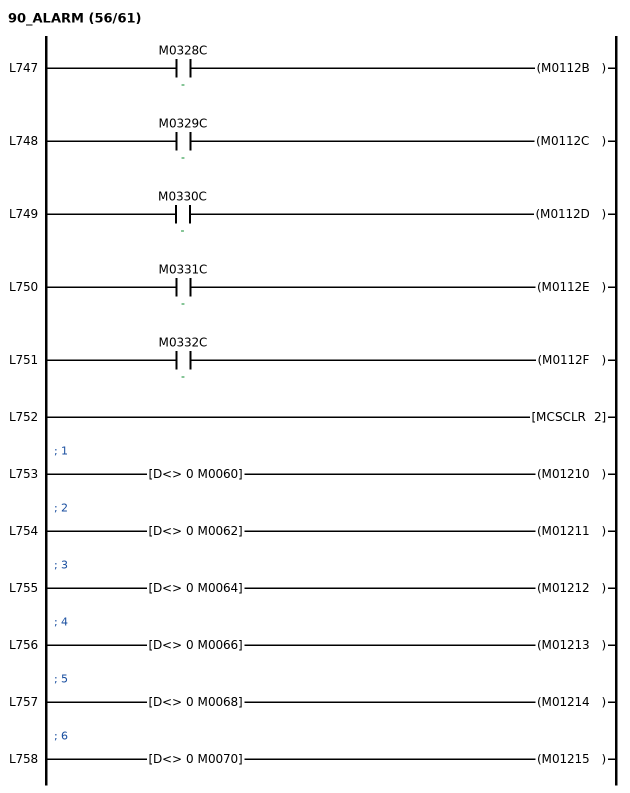
[picture p432: 90_ALARM rungs L747-L758]
; L747
LOAD      M0328C	// -
OUT       M0112B
; L748
LOAD      M0329C	// -
OUT       M0112C
; L749
LOAD      M0330C	// -
OUT       M0112D
; L750
LOAD      M0331C	// -
OUT       M0112E
; L751
LOAD      M0332C	// -
OUT       M0112F
; L752
MCSCLR    2
; L753
LOADD<>   0 M0060
OUT       M01210
// output comment: 1
; L754
LOADD<>   0 M0062
OUT       M01211
// output comment: 2
; L755
LOADD<>   0 M0064
OUT       M01212
// output comment: 3
; L756
LOADD<>   0 M0066
OUT       M01213
// output comment: 4
; L757
LOADD<>   0 M0068
OUT       M01214
// output comment: 5
; L758
LOADD<>   0 M0070
OUT       M01215
// output comment: 6

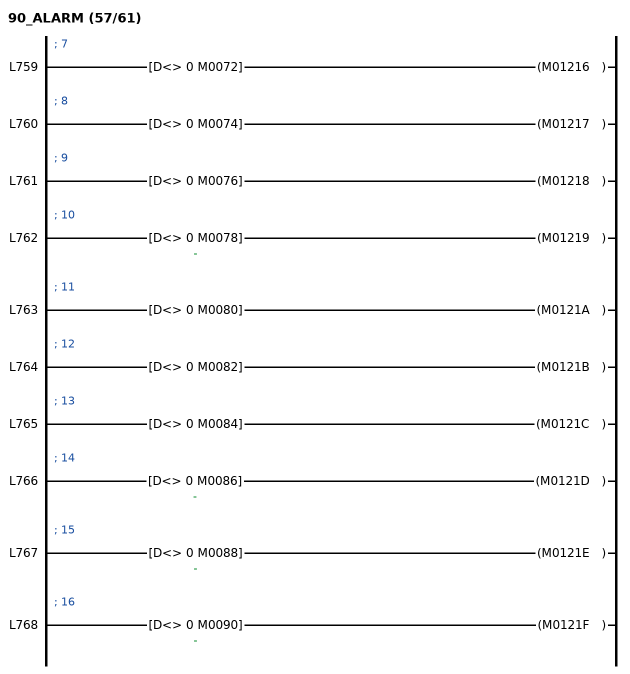
; L759
LOADD<>   0 M0072
OUT       M01216
// output comment: 7
; L760
LOADD<>   0 M0074
OUT       M01217
// output comment: 8
; L761
LOADD<>   0 M0076
OUT       M01218
// output comment: 9
; L762
LOADD<>   0 M0078	// -
OUT       M01219
// output comment: 10
; L763
LOADD<>   0 M0080
OUT       M0121A
// output comment: 11
; L764
LOADD<>   0 M0082
OUT       M0121B
// output comment: 12
; L765
LOADD<>   0 M0084
OUT       M0121C
// output comment: 13
; L766
LOADD<>   0 M0086	// -
OUT       M0121D
// output comment: 14
; L767
LOADD<>   0 M0088	// -
OUT       M0121E
// output comment: 15
; L768
LOADD<>   0 M0090	// -
OUT       M0121F
// output comment: 16

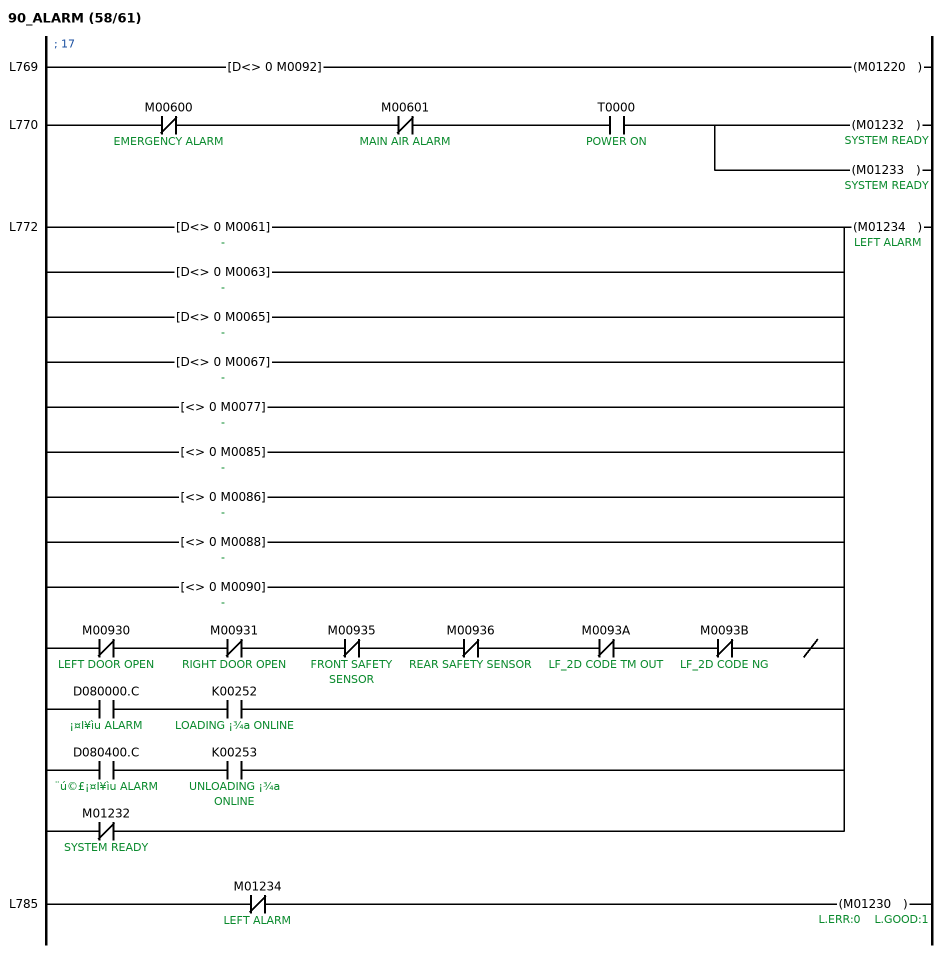
; L769
LOADD<>   0 M0092
OUT       M01220
// output comment: 17
; L770
LOAD NOT  M00600	// EMERGENCY ALARM
AND NOT   M00601	// MAIN AIR ALARM
AND       T0000	// POWER ON
OUT       M01232	// SYSTEM READY
OUT       M01233	// SYSTEM READY
; L772
LOADD<>   0 M0061	// -
ORD<>     0 M0063	// -
ORD<>     0 M0065	// -
ORD<>     0 M0067	// -
OR<>      0 M0077	// -
OR<>      0 M0085	// -
OR<>      0 M0086	// -
OR<>      0 M0088	// -
OR<>      0 M0090	// -
LOAD NOT  M00930	// LEFT DOOR OPEN
AND NOT   M00931	// RIGHT DOOR OPEN
AND NOT   M00935	// FRONT SAFETY SENSOR
AND NOT   M00936	// REAR SAFETY SENSOR
AND NOT   M0093A	// LF_2D CODE TM OUT
AND NOT   M0093B	// LF_2D CODE NG
NOT
OR LOAD
LOAD      D080000.C	// ¡¤I¥ìu ALARM
AND       K00252	// LOADING ¡¾a ONLINE
OR LOAD
LOAD      D080400.C	// ¨ú©£¡¤I¥ìu ALARM
AND       K00253	// UNLOADING ¡¾a ONLINE
OR LOAD
OR NOT    M01232	// SYSTEM READY
OUT       M01234	// LEFT ALARM
; L785
LOAD NOT  M01234	// LEFT ALARM
OUT       M01230	// L.ERR:0    L.GOOD:1

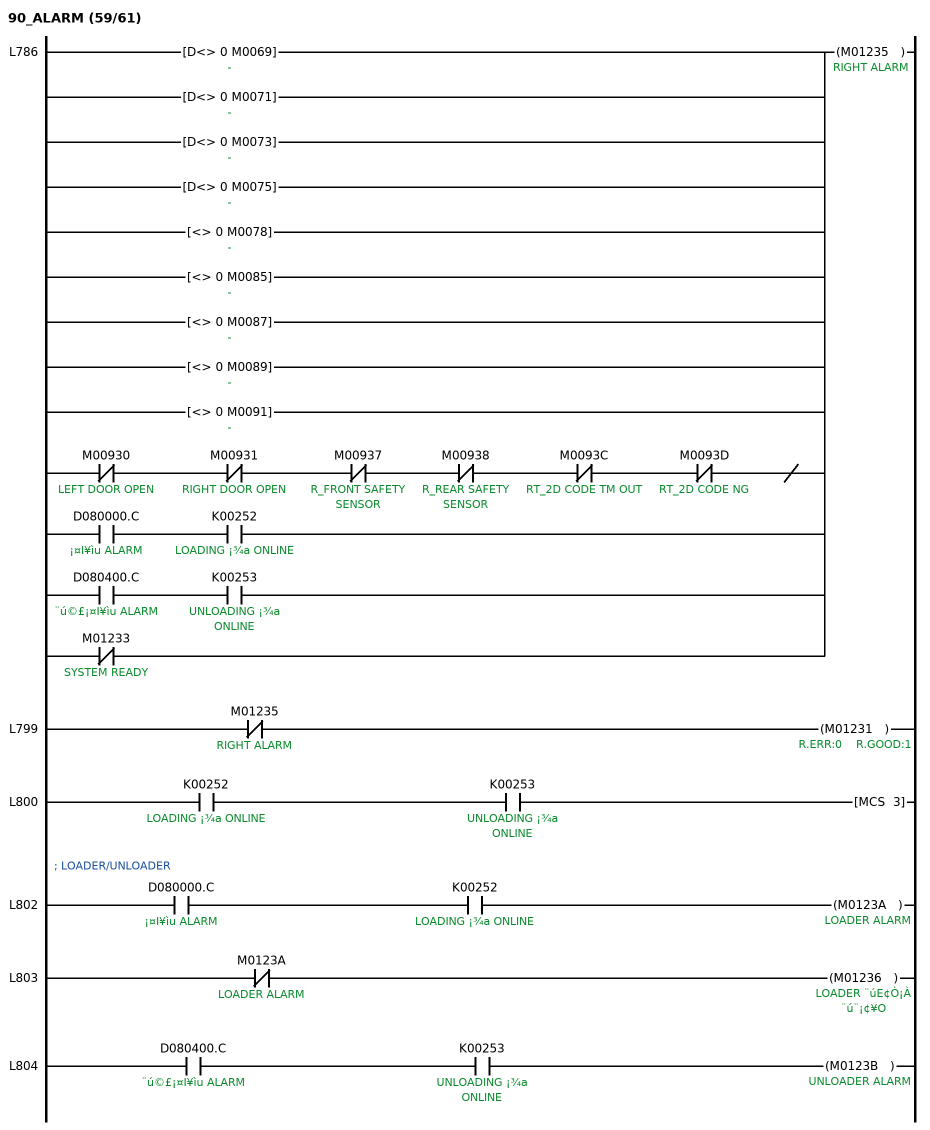
; L786
LOADD<>   0 M0069	// -
ORD<>     0 M0071	// -
ORD<>     0 M0073	// -
ORD<>     0 M0075	// -
OR<>      0 M0078	// -
OR<>      0 M0085	// -
OR<>      0 M0087	// -
OR<>      0 M0089	// -
OR<>      0 M0091	// -
LOAD NOT  M00930	// LEFT DOOR OPEN
AND NOT   M00931	// RIGHT DOOR OPEN
AND NOT   M00937	// R_FRONT SAFETY SENSOR
AND NOT   M00938	// R_REAR SAFETY SENSOR
AND NOT   M0093C	// RT_2D CODE TM OUT
AND NOT   M0093D	// RT_2D CODE NG
NOT
OR LOAD
LOAD      D080000.C	// ¡¤I¥ìu ALARM
AND       K00252	// LOADING ¡¾a ONLINE
OR LOAD
LOAD      D080400.C	// ¨ú©£¡¤I¥ìu ALARM
AND       K00253	// UNLOADING ¡¾a ONLINE
OR LOAD
OR NOT    M01233	// SYSTEM READY
OUT       M01235	// RIGHT ALARM
; L799
LOAD NOT  M01235	// RIGHT ALARM
OUT       M01231	// R.ERR:0    R.GOOD:1
; L800
LOAD      K00252	// LOADING ¡¾a ONLINE
AND       K00253	// UNLOADING ¡¾a ONLINE
MCS       3
// LOADER/UNLOADER
; L802
LOAD      D080000.C	// ¡¤I¥ìu ALARM
AND       K00252	// LOADING ¡¾a ONLINE
OUT       M0123A	// LOADER ALARM
; L803
LOAD NOT  M0123A	// LOADER ALARM
OUT       M01236	// LOADER ¨úE¢Ò¡À ¨ú¨¡¢¥O
; L804
LOAD      D080400.C	// ¨ú©£¡¤I¥ìu ALARM
AND       K00253	// UNLOADING ¡¾a ONLINE
OUT       M0123B	// UNLOADER ALARM

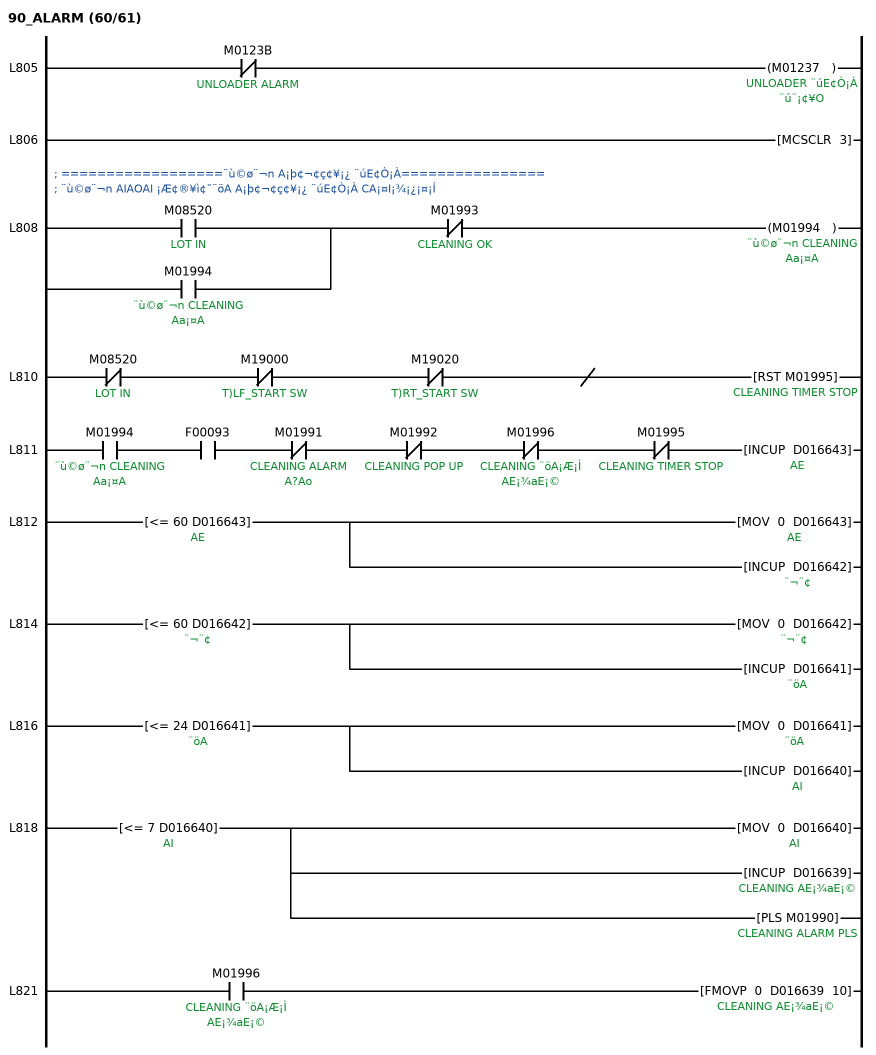
; L805
LOAD NOT  M0123B	// UNLOADER ALARM
OUT       M01237	// UNLOADER ¨úE¢Ò¡À ¨ú¨¡¢¥O
; L806
MCSCLR    3
// ==================¨ù©ø¨¬n A¡þ¢¬¢ç¢¥¡¿ ¨úE¢Ò¡À================
; L808
LOAD      M08520	// LOT IN
OR        M01994	// ¨ù©ø¨¬n CLEANING Aa¡¤A
AND NOT   M01993	// CLEANING OK
OUT       M01994	// ¨ù©ø¨¬n CLEANING Aa¡¤A
// output comment: ¨ù©ø¨¬n AIAOAI ¡Æ¢®¥ì¢¯¨öA A¡þ¢¬¢ç¢¥¡¿ ¨úE¢Ò¡À CA¡¤I¡¾¡¿¡¤¡Í
; L810
LOAD NOT  M08520	// LOT IN
AND NOT   M19000	// T)LF_START SW
AND NOT   M19020	// T)RT_START SW
NOT
RST       M01995	// CLEANING TIMER STOP
; L811
LOAD      M01994	// ¨ù©ø¨¬n CLEANING Aa¡¤A
AND       F00093
AND NOT   M01991	// CLEANING ALARM A?Ao
AND NOT   M01992	// CLEANING POP UP
AND NOT   M01996	// CLEANING ¨öA¡Æ¡Ì AE¡¾aE¡©
AND NOT   M01995	// CLEANING TIMER STOP
INCUP     D016643	// AE
; L812
LOAD<=    60 D016643	// AE
MOV       0 D016643	// AE
INCUP     D016642	// ¨¬¨¢
; L814
LOAD<=    60 D016642	// ¨¬¨¢
MOV       0 D016642	// ¨¬¨¢
INCUP     D016641	// ¨öA
; L816
LOAD<=    24 D016641	// ¨öA
MOV       0 D016641	// ¨öA
INCUP     D016640	// AI
; L818
LOAD<=    7 D016640	// AI
MOV       0 D016640	// AI
INCUP     D016639	// CLEANING AE¡¾aE¡©
OUTP      M01990	// CLEANING ALARM PLS
; L821
LOAD      M01996	// CLEANING ¨öA¡Æ¡Ì AE¡¾aE¡©
FMOVP     0 D016639 10	// CLEANING AE¡¾aE¡©

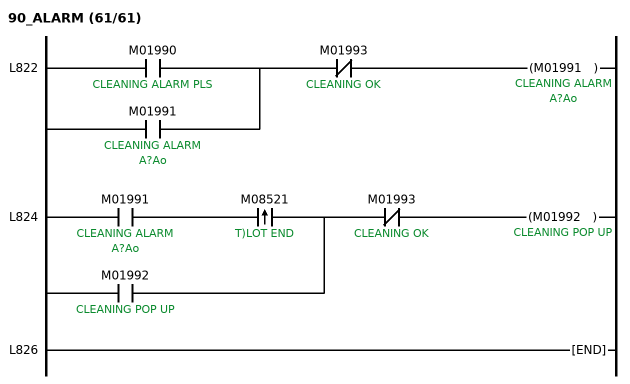
; L822
LOAD      M01990	// CLEANING ALARM PLS
OR        M01991	// CLEANING ALARM A?Ao
AND NOT   M01993	// CLEANING OK
OUT       M01991	// CLEANING ALARM A?Ao
; L824
LOAD      M01991	// CLEANING ALARM A?Ao
ANDP      M08521	// T)LOT END
OR        M01992	// CLEANING POP UP
AND NOT   M01993	// CLEANING OK
OUT       M01992	// CLEANING POP UP
; L826
END

PROGRAM 91_DEVICE_CHANGE (task: ¨ö¨¬A¥ì CA¡¤I¡¾¡¿¡¤¡Í)

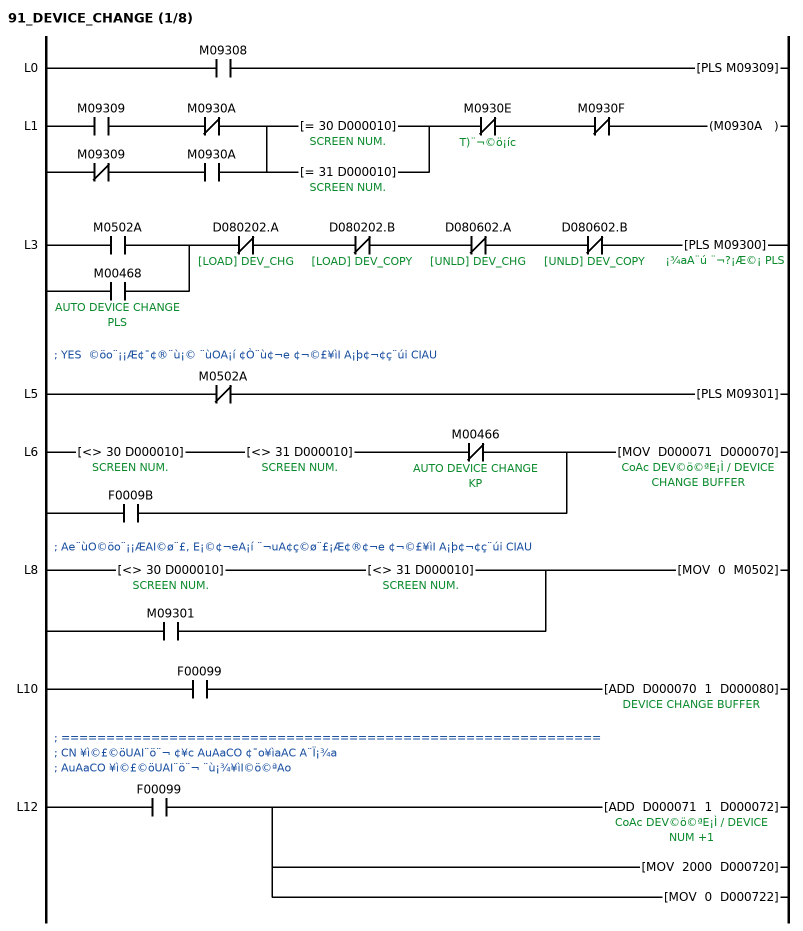
; L0
LOAD      M09308
OUTP      M09309
; L1
LOAD      M09309
AND NOT   M0930A
LOAD NOT  M09309
AND       M0930A
OR LOAD
LOAD=     30 D000010	// SCREEN NUM.
OR=       31 D000010	// SCREEN NUM.
AND LOAD
AND NOT   M0930E	// T)¨¬©ö¡íc
AND NOT   M0930F
OUT       M0930A
; L3
LOAD      M0502A
OR        M00468	// AUTO DEVICE CHANGE PLS
AND NOT   D080202.A	// [LOAD] DEV_CHG
AND NOT   D080202.B	// [LOAD] DEV_COPY
AND NOT   D080602.A	// [UNLD] DEV_CHG
AND NOT   D080602.B	// [UNLD] DEV_COPY
OUTP      M09300	// ¡¾aA¨ú ¨¬?¡Æ©¡ PLS
; L5
LOAD NOT  M0502A
OUTP      M09301
// output comment: YES  ©öo¨¡¡Æ¢¯¢®¨ù¡© ¨ùOA¡í ¢Ò¨ù¢¬e ¢¬©£¥ìI A¡þ¢¬¢ç¨úi CIAU
; L6
LOAD<>    30 D000010	// SCREEN NUM.
AND<>     31 D000010	// SCREEN NUM.
AND NOT   M00466	// AUTO DEVICE CHANGE KP
OR        F0009B
MOV       D000071 D000070	// CoAc DEV©ö©ªE¡Ì / DEVICE CHANGE BUFFER
; L8
LOAD<>    30 D000010	// SCREEN NUM.
AND<>     31 D000010	// SCREEN NUM.
OR        M09301
MOV       0 M0502
// output comment: Ae¨ùO©öo¨¡¡ÆAI©ø¨£, E¡©¢¬eA¡í ¨¬uA¢ç©ø¨£¡Æ¢®¢¬e ¢¬©£¥ìI A¡þ¢¬¢ç¨úi CIAU
; L10
LOAD      F00099
ADD       D000070 1 D000080	// DEVICE CHANGE BUFFER
// ============================================================
; L12
LOAD      F00099
ADD       D000071 1 D000072	// CoAc DEV©ö©ªE¡Ì / DEVICE NUM +1
MOV       2000 D000720
MOV       0 D000722
// output comment: CN ¥ì©£©öUAI¨ö¨¬ ¢¥c AuAaCO ¢¯o¥ìaAC A¨Ï¡¾a
// output comment: AuAaCO ¥ì©£©öUAI¨ö¨¬ ¨ù¡¾¥ìI©ö©ªAo

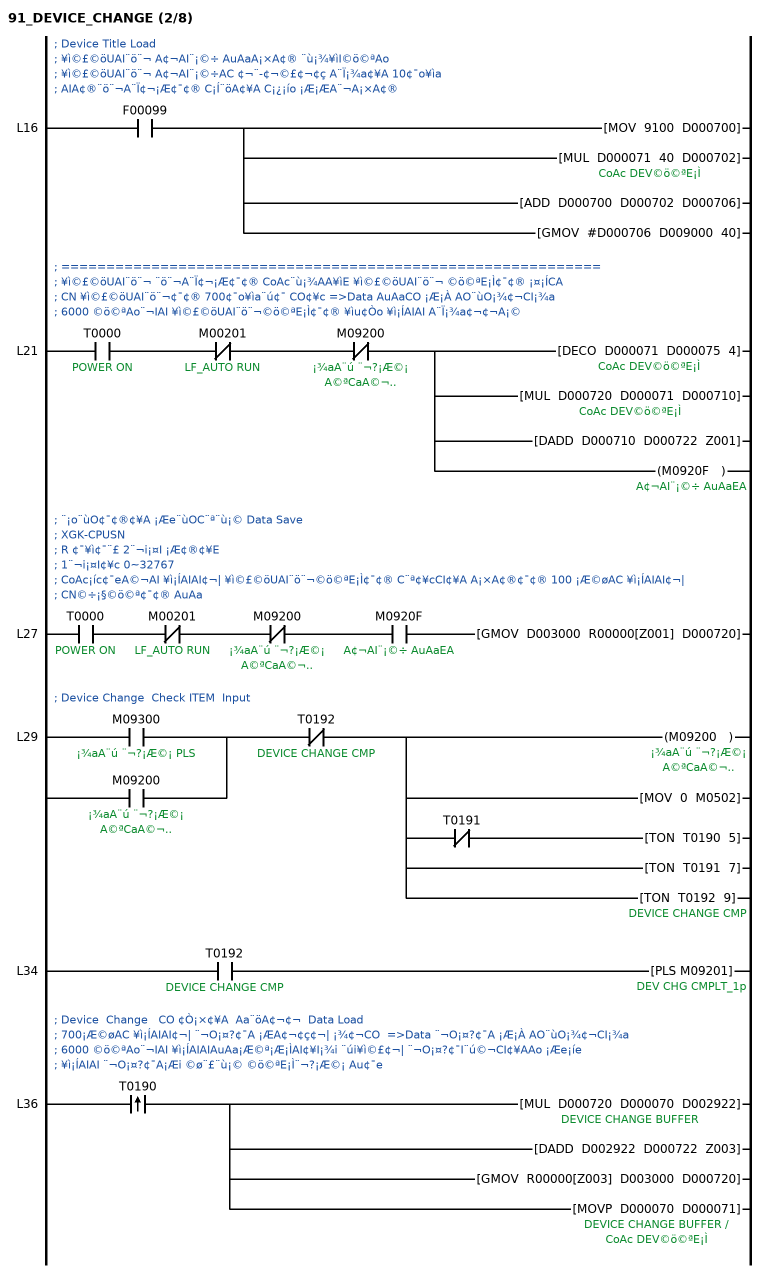
// Device Title Load
; L16
LOAD      F00099
MOV       9100 D000700
MUL       D000071 40 D000702	// CoAc DEV©ö©ªE¡Ì
ADD       D000700 D000702 D000706
GMOV      #D000706 D009000 40
// output comment: ¥ì©£©öUAI¨ö¨¬ A¢¬AI¨¡©÷ AuAaA¡×A¢® ¨ù¡¾¥ìI©ö©ªAo
// output comment: ¥ì©£©öUAI¨ö¨¬ A¢¬AI¨¡©÷AC ¢¬¨­¢¬©£¢¬¢ç A¨Ï¡¾a¢¥A 10¢¯o¥ìa
// output comment: AIA¢®¨ö¨¬A¨Ï¢¬¡Æ¢¯¢® C¡Í¨öA¢¥A C¡¿¡ío ¡Æ¡ÆA¨¬A¡×A¢®
// ============================================================
; L21
LOAD      T0000	// POWER ON
AND NOT   M00201	// LF_AUTO RUN
AND NOT   M09200	// ¡¾aA¨ú ¨¬?¡Æ©¡ A©ªCaA©¬..
DECO      D000071 D000075 4	// CoAc DEV©ö©ªE¡Ì
MUL       D000720 D000071 D000710	// CoAc DEV©ö©ªE¡Ì
DADD      D000710 D000722 Z001
OUT       M0920F	// A¢¬AI¨¡©÷ AuAaEA
// output comment: ¥ì©£©öUAI¨ö¨¬ ¨ö¨¬A¨Ï¢¬¡Æ¢¯¢® CoAc¨ù¡¾AA¥ìE ¥ì©£©öUAI¨ö¨¬ ©ö©ªE¡Ì¢¯¢® ¡¤¡ÍCA
// output comment: CN ¥ì©£©öUAI¨ö¨¬¢¯¢® 700¢¯o¥ìa¨ú¢¯ CO¢¥c =>Data AuAaCO ¡Æ¡À AO¨ùO¡¾¢¬CI¡¾a
// output comment: 6000 ©ö©ªAo¨¬IAI ¥ì©£©öUAI¨ö¨¬©ö©ªE¡Ì¢¯¢® ¥ìu¢Òo ¥ì¡ÍAIAI A¨Ï¡¾a¢¬¢¬A¡©
// ¨¡o¨ùO¢¯¢®¢¥A ¡Æe¨ùOC¨ª¨ù¡© Data Save
// XGK-CPUSN
// R ¢¯¥ì¢¯¨£ 2¨¬i¡¤I ¡Æ¢®¢¥E
// 1¨¬i¡¤I¢¥c 0~32767
; L27
LOAD      T0000	// POWER ON
AND NOT   M00201	// LF_AUTO RUN
AND NOT   M09200	// ¡¾aA¨ú ¨¬?¡Æ©¡ A©ªCaA©¬..
AND       M0920F	// A¢¬AI¨¡©÷ AuAaEA
GMOV      D003000 R00000[Z001] D000720
// output comment: CoAc¡íc¢¯eA©¬AI ¥ì¡ÍAIAI¢¬| ¥ì©£©öUAI¨ö¨¬©ö©ªE¡Ì¢¯¢® C¨ª¢¥cCI¢¥A A¡×A¢®¢¯¢® 100 ¡Æ©øAC ¥ì¡ÍAIAI¢¬| CN©÷¡§©ö©ª¢¯¢® AuAa
// Device Change  Check ITEM  Input
; L29
LOAD      M09300	// ¡¾aA¨ú ¨¬?¡Æ©¡ PLS
OR        M09200	// ¡¾aA¨ú ¨¬?¡Æ©¡ A©ªCaA©¬..
AND NOT   T0192	// DEVICE CHANGE CMP
OUT       M09200	// ¡¾aA¨ú ¨¬?¡Æ©¡ A©ªCaA©¬..
MOV       0 M0502
MPUSH
AND NOT   T0191
TON       T0190 5
MPOP
TON       T0191 7
TON       T0192 9	// DEVICE CHANGE CMP
; L34
LOAD      T0192	// DEVICE CHANGE CMP
OUTP      M09201	// DEV CHG CMPLT_1p
// Device  Change   CO ¢Ò¡×¢¥A  Aa¨öA¢¬¢¬  Data Load
; L36
LOADP     T0190
MUL       D000720 D000070 D002922	// DEVICE CHANGE BUFFER
DADD      D002922 D000722 Z003
GMOV      R00000[Z003] D003000 D000720
MOVP      D000070 D000071	// DEVICE CHANGE BUFFER / CoAc DEV©ö©ªE¡Ì
// output comment: 700¡Æ©øAC ¥ì¡ÍAIAI¢¬| ¨¬O¡¤?¢¯A ¡ÆA¢¬¢ç¢¬| ¡¾¢¬CO  =>Data ¨¬O¡¤?¢¯A ¡Æ¡À AO¨ùO¡¾¢¬CI¡¾a
// output comment: 6000 ©ö©ªAo¨¬IAI ¥ì¡ÍAIAIAuAa¡Æ©ª¡Æ¡ÌAI¢¥I¡¾i ¨úi¥ì©£¢¬| ¨¬O¡¤?¢¯I¨ú©¬CI¢¥AAo ¡Æe¡íe
// output comment: ¥ì¡ÍAIAI ¨¬O¡¤?¢¯A¡Æi ©ø¨£¨ù¡© ©ö©ªE¡Ì¨¬?¡Æ©¡ Au¢¯e

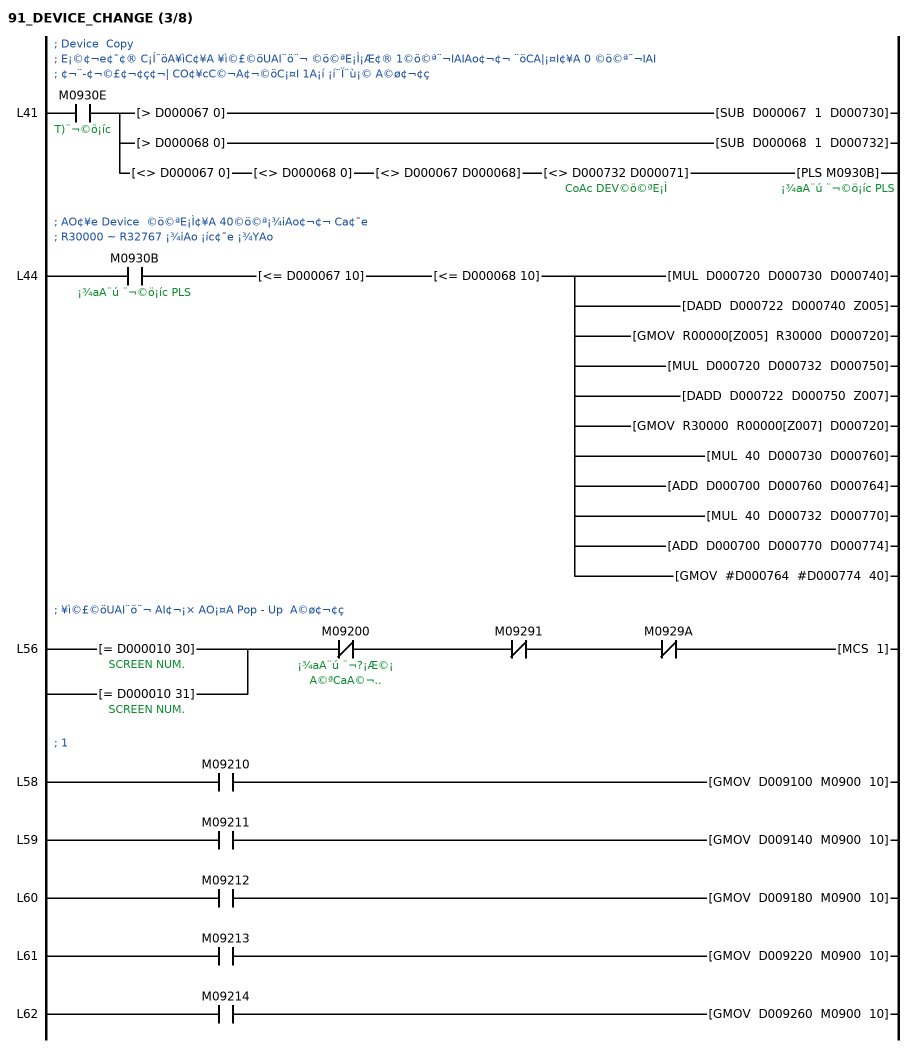
// Device  Copy
; L41
LOAD      M0930E	// T)¨¬©ö¡íc
MPUSH
AND>      D000067 0
SUB       D000067 1 D000730
MLOAD
AND>      D000068 0
SUB       D000068 1 D000732
MPOP
AND<>     D000067 0
AND<>     D000068 0
AND<>     D000067 D000068
AND<>     D000732 D000071	// CoAc DEV©ö©ªE¡Ì
OUTP      M0930B	// ¡¾aA¨ú ¨¬©ö¡íc PLS
// output comment: E¡©¢¬e¢¯¢® C¡Í¨öA¥ìC¢¥A ¥ì©£©öUAI¨ö¨¬ ©ö©ªE¡Ì¡Æ¢® 1©ö©ª¨¬IAIAo¢¬¢¬ ¨öCA|¡¤I¢¥A 0 ©ö©ª¨¬IAI
// output comment: ¢¬¨­¢¬©£¢¬¢ç¢¬| CO¢¥cC©¬A¢¬©öC¡¤I 1A¡í ¡í¨Ï¨ù¡© A©ø¢¬¢ç
; L44
LOAD      M0930B	// ¡¾aA¨ú ¨¬©ö¡íc PLS
AND<=     D000067 10
AND<=     D000068 10
MUL       D000720 D000730 D000740
DADD      D000722 D000740 Z005
GMOV      R00000[Z005] R30000 D000720
MUL       D000720 D000732 D000750
DADD      D000722 D000750 Z007
GMOV      R30000 R00000[Z007] D000720
MUL       40 D000730 D000760
ADD       D000700 D000760 D000764
MUL       40 D000732 D000770
ADD       D000700 D000770 D000774
GMOV      #D000764 #D000774 40
// output comment: AO¢¥e Device  ©ö©ªE¡Ì¢¥A 40©ö©ª¡¾iAo¢¬¢¬ Ca¢¯e
// output comment: R30000 ~ R32767 ¡¾iAo ¡íc¢¯e ¡¾YAo
// ¥ì©£©öUAI¨ö¨¬ AI¢¬¡× AO¡¤A Pop - Up  A©ø¢¬¢ç
; L56
LOAD=     D000010 30	// SCREEN NUM.
OR=       D000010 31	// SCREEN NUM.
AND NOT   M09200	// ¡¾aA¨ú ¨¬?¡Æ©¡ A©ªCaA©¬..
AND NOT   M09291
AND NOT   M0929A
MCS       1
; L58
LOAD      M09210
GMOV      D009100 M0900 10
// output comment: 1
; L59
LOAD      M09211
GMOV      D009140 M0900 10
; L60
LOAD      M09212
GMOV      D009180 M0900 10
; L61
LOAD      M09213
GMOV      D009220 M0900 10
; L62
LOAD      M09214
GMOV      D009260 M0900 10

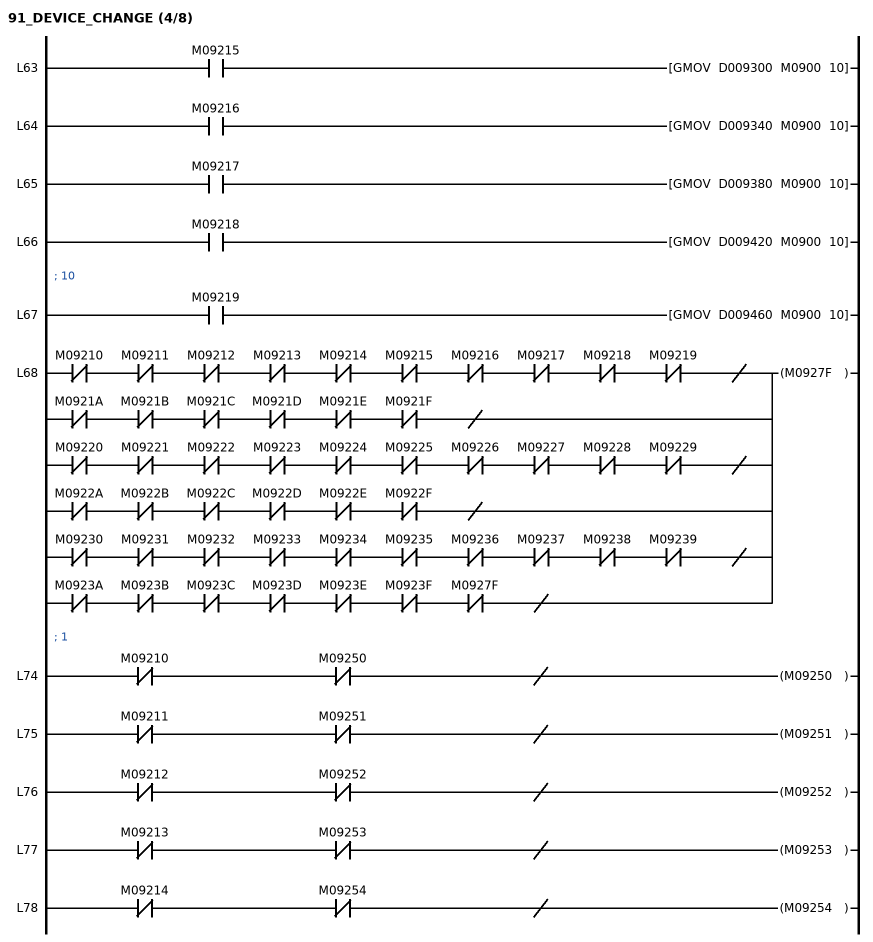
; L63
LOAD      M09215
GMOV      D009300 M0900 10
; L64
LOAD      M09216
GMOV      D009340 M0900 10
; L65
LOAD      M09217
GMOV      D009380 M0900 10
; L66
LOAD      M09218
GMOV      D009420 M0900 10
; L67
LOAD      M09219
GMOV      D009460 M0900 10
// output comment: 10
; L68
LOAD NOT  M09210
AND NOT   M09211
AND NOT   M09212
AND NOT   M09213
AND NOT   M09214
AND NOT   M09215
AND NOT   M09216
AND NOT   M09217
AND NOT   M09218
AND NOT   M09219
NOT
LOAD NOT  M0921A
AND NOT   M0921B
AND NOT   M0921C
AND NOT   M0921D
AND NOT   M0921E
AND NOT   M0921F
NOT
OR LOAD
LOAD NOT  M09220
AND NOT   M09221
AND NOT   M09222
AND NOT   M09223
AND NOT   M09224
AND NOT   M09225
AND NOT   M09226
AND NOT   M09227
AND NOT   M09228
AND NOT   M09229
NOT
OR LOAD
LOAD NOT  M0922A
AND NOT   M0922B
AND NOT   M0922C
AND NOT   M0922D
AND NOT   M0922E
AND NOT   M0922F
NOT
OR LOAD
LOAD NOT  M09230
AND NOT   M09231
AND NOT   M09232
AND NOT   M09233
AND NOT   M09234
AND NOT   M09235
AND NOT   M09236
AND NOT   M09237
AND NOT   M09238
AND NOT   M09239
NOT
OR LOAD
LOAD NOT  M0923A
AND NOT   M0923B
AND NOT   M0923C
AND NOT   M0923D
AND NOT   M0923E
AND NOT   M0923F
AND NOT   M0927F
NOT
OR LOAD
OUT       M0927F
; L74
LOAD NOT  M09210
AND NOT   M09250
NOT
OUT       M09250
// output comment: 1
; L75
LOAD NOT  M09211
AND NOT   M09251
NOT
OUT       M09251
; L76
LOAD NOT  M09212
AND NOT   M09252
NOT
OUT       M09252
; L77
LOAD NOT  M09213
AND NOT   M09253
NOT
OUT       M09253
; L78
LOAD NOT  M09214
AND NOT   M09254
NOT
OUT       M09254

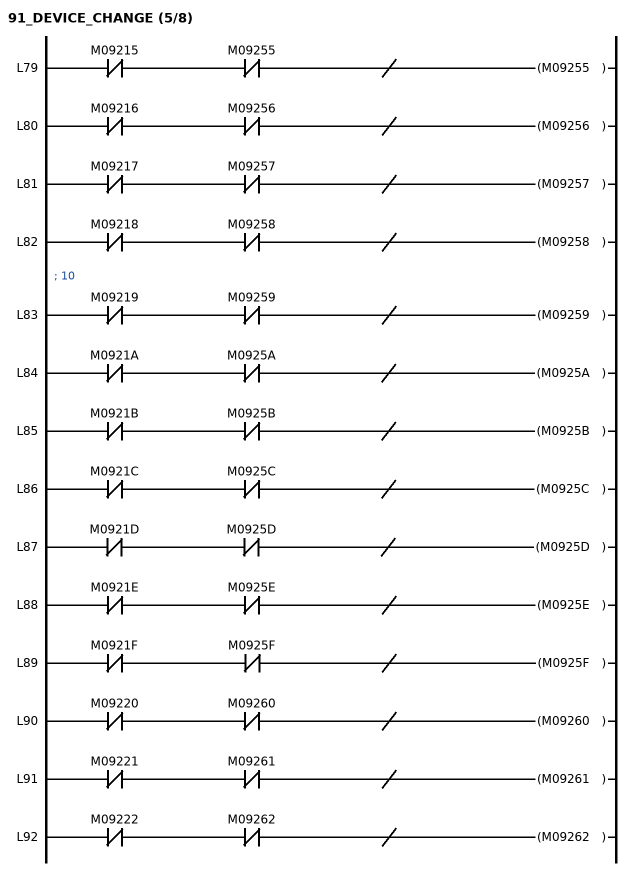
; L79
LOAD NOT  M09215
AND NOT   M09255
NOT
OUT       M09255
; L80
LOAD NOT  M09216
AND NOT   M09256
NOT
OUT       M09256
; L81
LOAD NOT  M09217
AND NOT   M09257
NOT
OUT       M09257
; L82
LOAD NOT  M09218
AND NOT   M09258
NOT
OUT       M09258
; L83
LOAD NOT  M09219
AND NOT   M09259
NOT
OUT       M09259
// output comment: 10
; L84
LOAD NOT  M0921A
AND NOT   M0925A
NOT
OUT       M0925A
; L85
LOAD NOT  M0921B
AND NOT   M0925B
NOT
OUT       M0925B
; L86
LOAD NOT  M0921C
AND NOT   M0925C
NOT
OUT       M0925C
; L87
LOAD NOT  M0921D
AND NOT   M0925D
NOT
OUT       M0925D
; L88
LOAD NOT  M0921E
AND NOT   M0925E
NOT
OUT       M0925E
; L89
LOAD NOT  M0921F
AND NOT   M0925F
NOT
OUT       M0925F
; L90
LOAD NOT  M09220
AND NOT   M09260
NOT
OUT       M09260
; L91
LOAD NOT  M09221
AND NOT   M09261
NOT
OUT       M09261
; L92
LOAD NOT  M09222
AND NOT   M09262
NOT
OUT       M09262

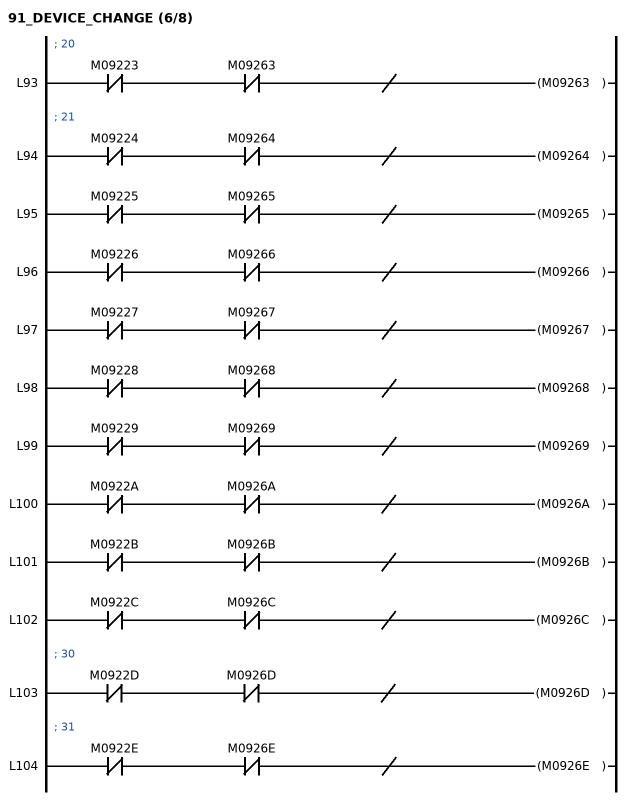
; L93
LOAD NOT  M09223
AND NOT   M09263
NOT
OUT       M09263
// output comment: 20
; L94
LOAD NOT  M09224
AND NOT   M09264
NOT
OUT       M09264
// output comment: 21
; L95
LOAD NOT  M09225
AND NOT   M09265
NOT
OUT       M09265
; L96
LOAD NOT  M09226
AND NOT   M09266
NOT
OUT       M09266
; L97
LOAD NOT  M09227
AND NOT   M09267
NOT
OUT       M09267
; L98
LOAD NOT  M09228
AND NOT   M09268
NOT
OUT       M09268
; L99
LOAD NOT  M09229
AND NOT   M09269
NOT
OUT       M09269
; L100
LOAD NOT  M0922A
AND NOT   M0926A
NOT
OUT       M0926A
; L101
LOAD NOT  M0922B
AND NOT   M0926B
NOT
OUT       M0926B
; L102
LOAD NOT  M0922C
AND NOT   M0926C
NOT
OUT       M0926C
; L103
LOAD NOT  M0922D
AND NOT   M0926D
NOT
OUT       M0926D
// output comment: 30
; L104
LOAD NOT  M0922E
AND NOT   M0926E
NOT
OUT       M0926E
// output comment: 31

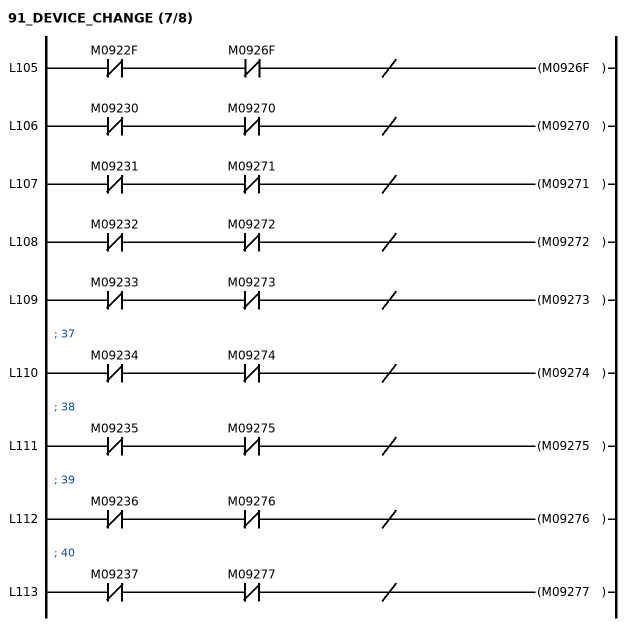
; L105
LOAD NOT  M0922F
AND NOT   M0926F
NOT
OUT       M0926F
; L106
LOAD NOT  M09230
AND NOT   M09270
NOT
OUT       M09270
; L107
LOAD NOT  M09231
AND NOT   M09271
NOT
OUT       M09271
; L108
LOAD NOT  M09232
AND NOT   M09272
NOT
OUT       M09272
; L109
LOAD NOT  M09233
AND NOT   M09273
NOT
OUT       M09273
; L110
LOAD NOT  M09234
AND NOT   M09274
NOT
OUT       M09274
// output comment: 37
; L111
LOAD NOT  M09235
AND NOT   M09275
NOT
OUT       M09275
// output comment: 38
; L112
LOAD NOT  M09236
AND NOT   M09276
NOT
OUT       M09276
// output comment: 39
; L113
LOAD NOT  M09237
AND NOT   M09277
NOT
OUT       M09277
// output comment: 40

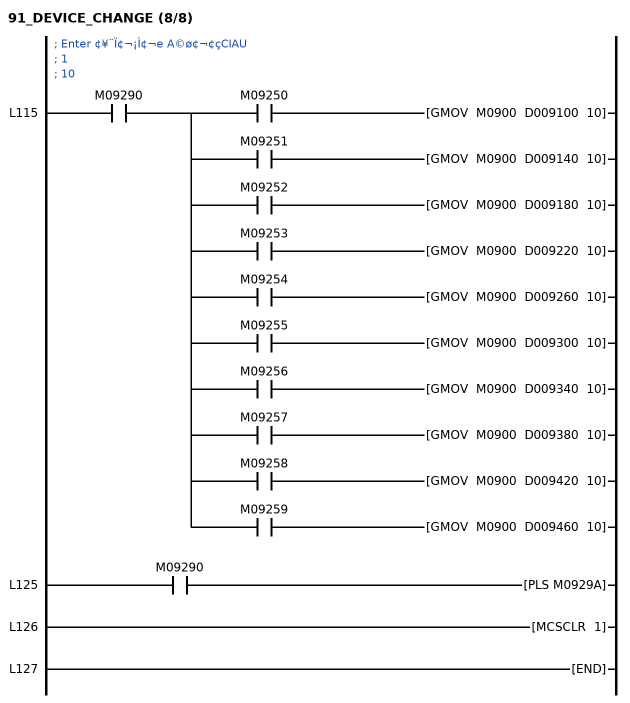
// Enter ¢¥¨Ï¢¬¡Ì¢¬e A©ø¢¬¢çCIAU
; L115
LOAD      M09290
MPUSH
AND       M09250
GMOV      M0900 D009100 10
MLOAD
AND       M09251
GMOV      M0900 D009140 10
MLOAD
AND       M09252
GMOV      M0900 D009180 10
MLOAD
AND       M09253
GMOV      M0900 D009220 10
MLOAD
AND       M09254
GMOV      M0900 D009260 10
MLOAD
AND       M09255
GMOV      M0900 D009300 10
MLOAD
AND       M09256
GMOV      M0900 D009340 10
MLOAD
AND       M09257
GMOV      M0900 D009380 10
MLOAD
AND       M09258
GMOV      M0900 D009420 10
MPOP
AND       M09259
GMOV      M0900 D009460 10
// output comment: 1
// output comment: 10
; L125
LOAD      M09290
OUTP      M0929A
; L126
MCSCLR    1
; L127
END

PROGRAM 92_ALARM_SCR (task: ¨ö¨¬A¥ì CA¡¤I¡¾¡¿¡¤¡Í)

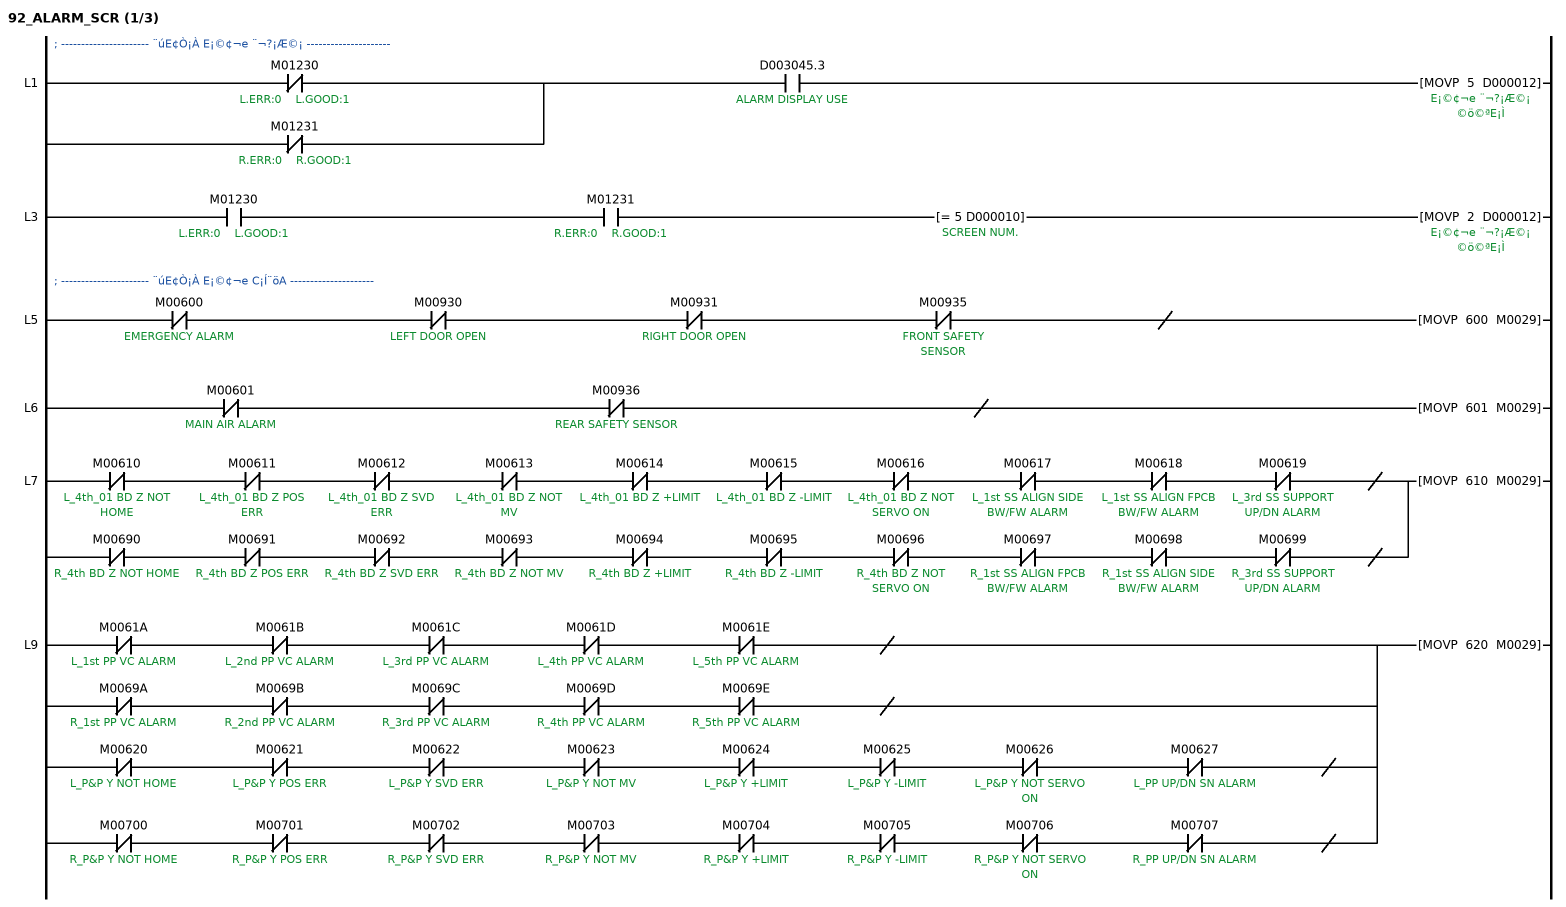
// ---------------------- ¨úE¢Ò¡À E¡©¢¬e ¨¬?¡Æ©¡ ---------------------
; L1
LOAD NOT  M01230	// L.ERR:0    L.GOOD:1
OR NOT    M01231	// R.ERR:0    R.GOOD:1
AND       D003045.3	// ALARM DISPLAY USE
MOVP      5 D000012	// E¡©¢¬e ¨¬?¡Æ©¡ ©ö©ªE¡Ì
; L3
LOAD      M01230	// L.ERR:0    L.GOOD:1
AND       M01231	// R.ERR:0    R.GOOD:1
AND=      5 D000010	// SCREEN NUM.
MOVP      2 D000012	// E¡©¢¬e ¨¬?¡Æ©¡ ©ö©ªE¡Ì
// ---------------------- ¨úE¢Ò¡À E¡©¢¬e C¡Í¨öA ---------------------
; L5
LOAD NOT  M00600	// EMERGENCY ALARM
AND NOT   M00930	// LEFT DOOR OPEN
AND NOT   M00931	// RIGHT DOOR OPEN
AND NOT   M00935	// FRONT SAFETY SENSOR
NOT
MOVP      600 M0029
; L6
LOAD NOT  M00601	// MAIN AIR ALARM
AND NOT   M00936	// REAR SAFETY SENSOR
NOT
MOVP      601 M0029
; L7
LOAD NOT  M00610	// L_4th_01 BD Z NOT HOME
AND NOT   M00611	// L_4th_01 BD Z POS ERR
AND NOT   M00612	// L_4th_01 BD Z SVD ERR
AND NOT   M00613	// L_4th_01 BD Z NOT MV
AND NOT   M00614	// L_4th_01 BD Z +LIMIT
AND NOT   M00615	// L_4th_01 BD Z -LIMIT
AND NOT   M00616	// L_4th_01 BD Z NOT SERVO ON
AND NOT   M00617	// L_1st SS ALIGN SIDE BW/FW ALARM
AND NOT   M00618	// L_1st SS ALIGN FPCB BW/FW ALARM
AND NOT   M00619	// L_3rd SS SUPPORT UP/DN ALARM
NOT
LOAD NOT  M00690	// R_4th BD Z NOT HOME
AND NOT   M00691	// R_4th BD Z POS ERR
AND NOT   M00692	// R_4th BD Z SVD ERR
AND NOT   M00693	// R_4th BD Z NOT MV
AND NOT   M00694	// R_4th BD Z +LIMIT
AND NOT   M00695	// R_4th BD Z -LIMIT
AND NOT   M00696	// R_4th BD Z NOT SERVO ON
AND NOT   M00697	// R_1st SS ALIGN FPCB BW/FW ALARM
AND NOT   M00698	// R_1st SS ALIGN SIDE BW/FW ALARM
AND NOT   M00699	// R_3rd SS SUPPORT UP/DN ALARM
NOT
OR LOAD
MOVP      610 M0029
; L9
LOAD NOT  M0061A	// L_1st PP VC ALARM
AND NOT   M0061B	// L_2nd PP VC ALARM
AND NOT   M0061C	// L_3rd PP VC ALARM
AND NOT   M0061D	// L_4th PP VC ALARM
AND NOT   M0061E	// L_5th PP VC ALARM
NOT
LOAD NOT  M0069A	// R_1st PP VC ALARM
AND NOT   M0069B	// R_2nd PP VC ALARM
AND NOT   M0069C	// R_3rd PP VC ALARM
AND NOT   M0069D	// R_4th PP VC ALARM
AND NOT   M0069E	// R_5th PP VC ALARM
NOT
OR LOAD
LOAD NOT  M00620	// L_P&P Y NOT HOME
AND NOT   M00621	// L_P&P Y POS ERR
AND NOT   M00622	// L_P&P Y SVD ERR
AND NOT   M00623	// L_P&P Y NOT MV
AND NOT   M00624	// L_P&P Y +LIMIT
AND NOT   M00625	// L_P&P Y -LIMIT
AND NOT   M00626	// L_P&P Y NOT SERVO ON
AND NOT   M00627	// L_PP UP/DN SN ALARM
NOT
OR LOAD
LOAD NOT  M00700	// R_P&P Y NOT HOME
AND NOT   M00701	// R_P&P Y POS ERR
AND NOT   M00702	// R_P&P Y SVD ERR
AND NOT   M00703	// R_P&P Y NOT MV
AND NOT   M00704	// R_P&P Y +LIMIT
AND NOT   M00705	// R_P&P Y -LIMIT
AND NOT   M00706	// R_P&P Y NOT SERVO ON
AND NOT   M00707	// R_PP UP/DN SN ALARM
NOT
OR LOAD
MOVP      620 M0029

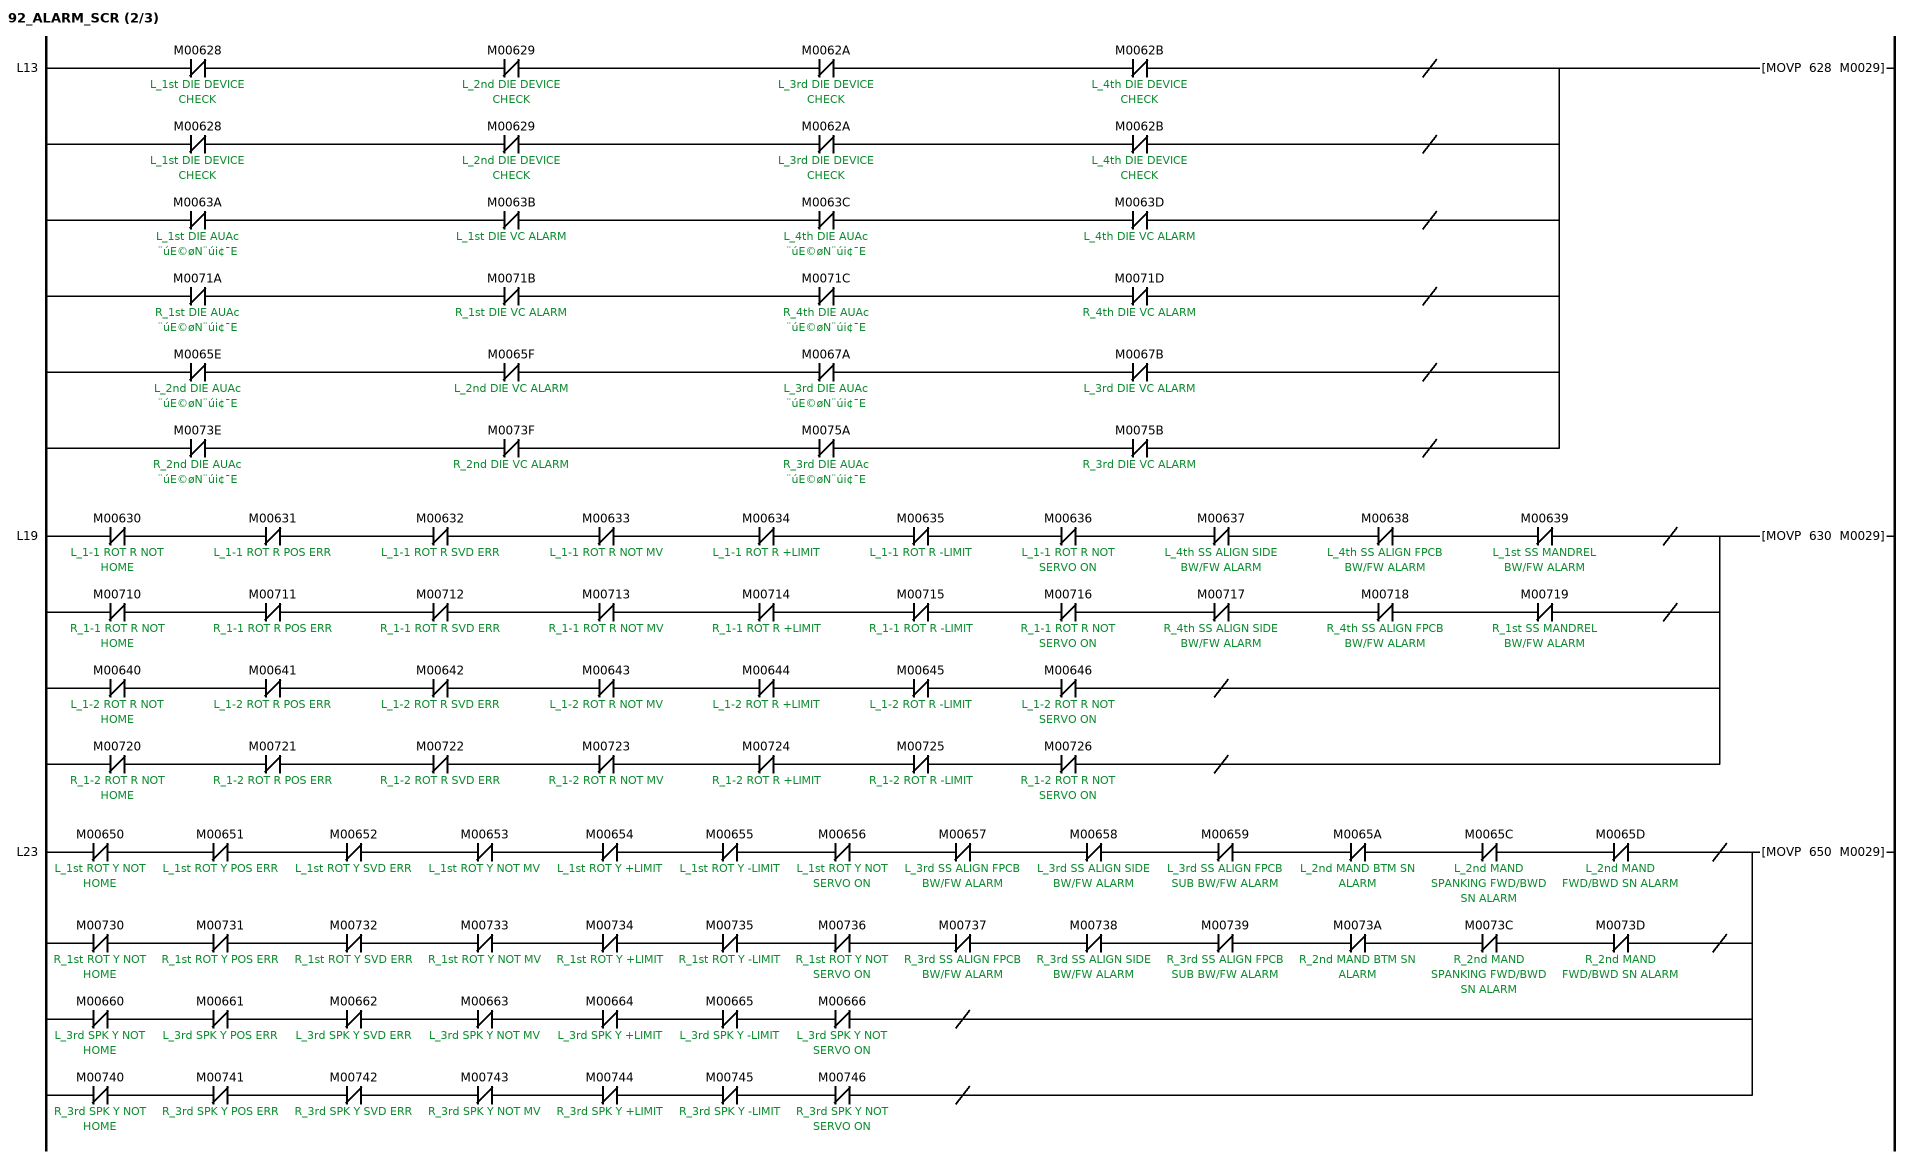
; L13
LOAD NOT  M00628	// L_1st DIE DEVICE CHECK
AND NOT   M00629	// L_2nd DIE DEVICE CHECK
AND NOT   M0062A	// L_3rd DIE DEVICE CHECK
AND NOT   M0062B	// L_4th DIE DEVICE CHECK
NOT
LOAD NOT  M00628	// L_1st DIE DEVICE CHECK
AND NOT   M00629	// L_2nd DIE DEVICE CHECK
AND NOT   M0062A	// L_3rd DIE DEVICE CHECK
AND NOT   M0062B	// L_4th DIE DEVICE CHECK
NOT
OR LOAD
LOAD NOT  M0063A	// L_1st DIE AUAc ¨úE©øN¨úi¢¯E
AND NOT   M0063B	// L_1st DIE VC ALARM
AND NOT   M0063C	// L_4th DIE AUAc ¨úE©øN¨úi¢¯E
AND NOT   M0063D	// L_4th DIE VC ALARM
NOT
OR LOAD
LOAD NOT  M0071A	// R_1st DIE AUAc ¨úE©øN¨úi¢¯E
AND NOT   M0071B	// R_1st DIE VC ALARM
AND NOT   M0071C	// R_4th DIE AUAc ¨úE©øN¨úi¢¯E
AND NOT   M0071D	// R_4th DIE VC ALARM
NOT
OR LOAD
LOAD NOT  M0065E	// L_2nd DIE AUAc ¨úE©øN¨úi¢¯E
AND NOT   M0065F	// L_2nd DIE VC ALARM
AND NOT   M0067A	// L_3rd DIE AUAc ¨úE©øN¨úi¢¯E
AND NOT   M0067B	// L_3rd DIE VC ALARM
NOT
OR LOAD
LOAD NOT  M0073E	// R_2nd DIE AUAc ¨úE©øN¨úi¢¯E
AND NOT   M0073F	// R_2nd DIE VC ALARM
AND NOT   M0075A	// R_3rd DIE AUAc ¨úE©øN¨úi¢¯E
AND NOT   M0075B	// R_3rd DIE VC ALARM
NOT
OR LOAD
MOVP      628 M0029
; L19
LOAD NOT  M00630	// L_1-1 ROT R NOT HOME
AND NOT   M00631	// L_1-1 ROT R POS ERR
AND NOT   M00632	// L_1-1 ROT R SVD ERR
AND NOT   M00633	// L_1-1 ROT R NOT MV
AND NOT   M00634	// L_1-1 ROT R +LIMIT
AND NOT   M00635	// L_1-1 ROT R -LIMIT
AND NOT   M00636	// L_1-1 ROT R NOT SERVO ON
AND NOT   M00637	// L_4th SS ALIGN SIDE BW/FW ALARM
AND NOT   M00638	// L_4th SS ALIGN FPCB BW/FW ALARM
AND NOT   M00639	// L_1st SS MANDREL BW/FW ALARM
NOT
LOAD NOT  M00710	// R_1-1 ROT R NOT HOME
AND NOT   M00711	// R_1-1 ROT R POS ERR
AND NOT   M00712	// R_1-1 ROT R SVD ERR
AND NOT   M00713	// R_1-1 ROT R NOT MV
AND NOT   M00714	// R_1-1 ROT R +LIMIT
AND NOT   M00715	// R_1-1 ROT R -LIMIT
AND NOT   M00716	// R_1-1 ROT R NOT SERVO ON
AND NOT   M00717	// R_4th SS ALIGN SIDE BW/FW ALARM
AND NOT   M00718	// R_4th SS ALIGN FPCB BW/FW ALARM
AND NOT   M00719	// R_1st SS MANDREL BW/FW ALARM
NOT
OR LOAD
LOAD NOT  M00640	// L_1-2 ROT R NOT HOME
AND NOT   M00641	// L_1-2 ROT R POS ERR
AND NOT   M00642	// L_1-2 ROT R SVD ERR
AND NOT   M00643	// L_1-2 ROT R NOT MV
AND NOT   M00644	// L_1-2 ROT R +LIMIT
AND NOT   M00645	// L_1-2 ROT R -LIMIT
AND NOT   M00646	// L_1-2 ROT R NOT SERVO ON
NOT
OR LOAD
LOAD NOT  M00720	// R_1-2 ROT R NOT HOME
AND NOT   M00721	// R_1-2 ROT R POS ERR
AND NOT   M00722	// R_1-2 ROT R SVD ERR
AND NOT   M00723	// R_1-2 ROT R NOT MV
AND NOT   M00724	// R_1-2 ROT R +LIMIT
AND NOT   M00725	// R_1-2 ROT R -LIMIT
AND NOT   M00726	// R_1-2 ROT R NOT SERVO ON
NOT
OR LOAD
MOVP      630 M0029
; L23
LOAD NOT  M00650	// L_1st ROT Y NOT HOME
AND NOT   M00651	// L_1st ROT Y POS ERR
AND NOT   M00652	// L_1st ROT Y SVD ERR
AND NOT   M00653	// L_1st ROT Y NOT MV
AND NOT   M00654	// L_1st ROT Y +LIMIT
AND NOT   M00655	// L_1st ROT Y -LIMIT
AND NOT   M00656	// L_1st ROT Y NOT SERVO ON
AND NOT   M00657	// L_3rd SS ALIGN FPCB BW/FW ALARM
AND NOT   M00658	// L_3rd SS ALIGN SIDE BW/FW ALARM
AND NOT   M00659	// L_3rd SS ALIGN FPCB SUB BW/FW ALARM
AND NOT   M0065A	// L_2nd MAND BTM SN ALARM
AND NOT   M0065C	// L_2nd MAND SPANKING FWD/BWD SN ALARM
AND NOT   M0065D	// L_2nd MAND FWD/BWD SN ALARM
NOT
LOAD NOT  M00730	// R_1st ROT Y NOT HOME
AND NOT   M00731	// R_1st ROT Y POS ERR
AND NOT   M00732	// R_1st ROT Y SVD ERR
AND NOT   M00733	// R_1st ROT Y NOT MV
AND NOT   M00734	// R_1st ROT Y +LIMIT
AND NOT   M00735	// R_1st ROT Y -LIMIT
AND NOT   M00736	// R_1st ROT Y NOT SERVO ON
AND NOT   M00737	// R_3rd SS ALIGN FPCB BW/FW ALARM
AND NOT   M00738	// R_3rd SS ALIGN SIDE BW/FW ALARM
AND NOT   M00739	// R_3rd SS ALIGN FPCB SUB BW/FW ALARM
AND NOT   M0073A	// R_2nd MAND BTM SN ALARM
AND NOT   M0073C	// R_2nd MAND SPANKING FWD/BWD SN ALARM
AND NOT   M0073D	// R_2nd MAND FWD/BWD SN ALARM
NOT
OR LOAD
LOAD NOT  M00660	// L_3rd SPK Y NOT HOME
AND NOT   M00661	// L_3rd SPK Y POS ERR
AND NOT   M00662	// L_3rd SPK Y SVD ERR
AND NOT   M00663	// L_3rd SPK Y NOT MV
AND NOT   M00664	// L_3rd SPK Y +LIMIT
AND NOT   M00665	// L_3rd SPK Y -LIMIT
AND NOT   M00666	// L_3rd SPK Y NOT SERVO ON
NOT
OR LOAD
LOAD NOT  M00740	// R_3rd SPK Y NOT HOME
AND NOT   M00741	// R_3rd SPK Y POS ERR
AND NOT   M00742	// R_3rd SPK Y SVD ERR
AND NOT   M00743	// R_3rd SPK Y NOT MV
AND NOT   M00744	// R_3rd SPK Y +LIMIT
AND NOT   M00745	// R_3rd SPK Y -LIMIT
AND NOT   M00746	// R_3rd SPK Y NOT SERVO ON
NOT
OR LOAD
MOVP      650 M0029

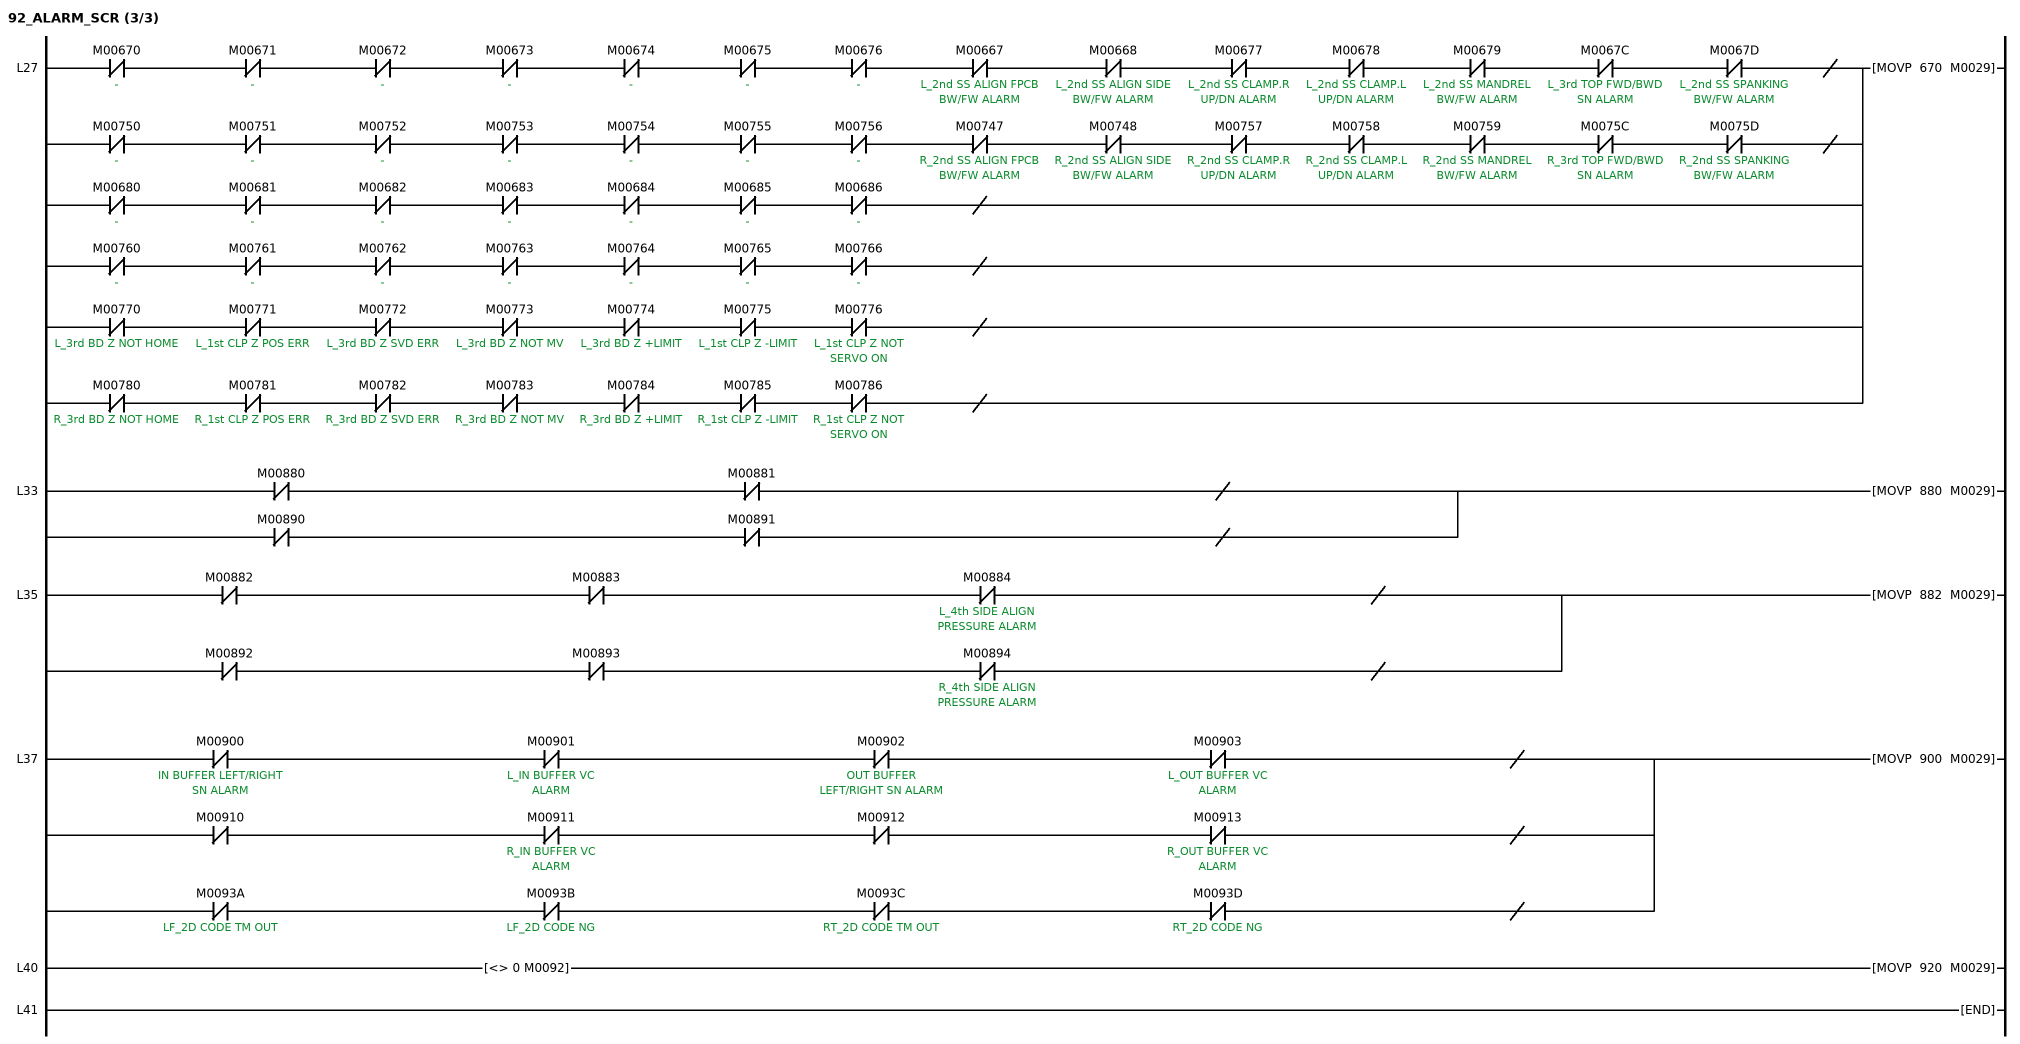
; L27
LOAD NOT  M00670	// -
AND NOT   M00671	// -
AND NOT   M00672	// -
AND NOT   M00673	// -
AND NOT   M00674	// -
AND NOT   M00675	// -
AND NOT   M00676	// -
AND NOT   M00667	// L_2nd SS ALIGN FPCB BW/FW ALARM
AND NOT   M00668	// L_2nd SS ALIGN SIDE BW/FW ALARM
AND NOT   M00677	// L_2nd SS CLAMP.R UP/DN ALARM
AND NOT   M00678	// L_2nd SS CLAMP.L UP/DN ALARM
AND NOT   M00679	// L_2nd SS MANDREL BW/FW ALARM
AND NOT   M0067C	// L_3rd TOP FWD/BWD SN ALARM
AND NOT   M0067D	// L_2nd SS SPANKING BW/FW ALARM
NOT
LOAD NOT  M00750	// -
AND NOT   M00751	// -
AND NOT   M00752	// -
AND NOT   M00753	// -
AND NOT   M00754	// -
AND NOT   M00755	// -
AND NOT   M00756	// -
AND NOT   M00747	// R_2nd SS ALIGN FPCB BW/FW ALARM
AND NOT   M00748	// R_2nd SS ALIGN SIDE BW/FW ALARM
AND NOT   M00757	// R_2nd SS CLAMP.R UP/DN ALARM
AND NOT   M00758	// R_2nd SS CLAMP.L UP/DN ALARM
AND NOT   M00759	// R_2nd SS MANDREL BW/FW ALARM
AND NOT   M0075C	// R_3rd TOP FWD/BWD SN ALARM
AND NOT   M0075D	// R_2nd SS SPANKING BW/FW ALARM
NOT
OR LOAD
LOAD NOT  M00680	// -
AND NOT   M00681	// -
AND NOT   M00682	// -
AND NOT   M00683	// -
AND NOT   M00684	// -
AND NOT   M00685	// -
AND NOT   M00686	// -
NOT
OR LOAD
LOAD NOT  M00760	// -
AND NOT   M00761	// -
AND NOT   M00762	// -
AND NOT   M00763	// -
AND NOT   M00764	// -
AND NOT   M00765	// -
AND NOT   M00766	// -
NOT
OR LOAD
LOAD NOT  M00770	// L_3rd BD Z NOT HOME
AND NOT   M00771	// L_1st CLP Z POS ERR
AND NOT   M00772	// L_3rd BD Z SVD ERR
AND NOT   M00773	// L_3rd BD Z NOT MV
AND NOT   M00774	// L_3rd BD Z +LIMIT
AND NOT   M00775	// L_1st CLP Z -LIMIT
AND NOT   M00776	// L_1st CLP Z NOT SERVO ON
NOT
OR LOAD
LOAD NOT  M00780	// R_3rd BD Z NOT HOME
AND NOT   M00781	// R_1st CLP Z POS ERR
AND NOT   M00782	// R_3rd BD Z SVD ERR
AND NOT   M00783	// R_3rd BD Z NOT MV
AND NOT   M00784	// R_3rd BD Z +LIMIT
AND NOT   M00785	// R_1st CLP Z -LIMIT
AND NOT   M00786	// R_1st CLP Z NOT SERVO ON
NOT
OR LOAD
MOVP      670 M0029
; L33
LOAD NOT  M00880
AND NOT   M00881
NOT
LOAD NOT  M00890
AND NOT   M00891
NOT
OR LOAD
MOVP      880 M0029
; L35
LOAD NOT  M00882
AND NOT   M00883
AND NOT   M00884	// L_4th SIDE ALIGN PRESSURE ALARM
NOT
LOAD NOT  M00892
AND NOT   M00893
AND NOT   M00894	// R_4th SIDE ALIGN PRESSURE ALARM
NOT
OR LOAD
MOVP      882 M0029
; L37
LOAD NOT  M00900	// IN BUFFER LEFT/RIGHT SN ALARM
AND NOT   M00901	// L_IN BUFFER VC ALARM
AND NOT   M00902	// OUT BUFFER LEFT/RIGHT SN ALARM
AND NOT   M00903	// L_OUT BUFFER VC ALARM
NOT
LOAD NOT  M00910
AND NOT   M00911	// R_IN BUFFER VC ALARM
AND NOT   M00912
AND NOT   M00913	// R_OUT BUFFER VC ALARM
NOT
OR LOAD
LOAD NOT  M0093A	// LF_2D CODE TM OUT
AND NOT   M0093B	// LF_2D CODE NG
AND NOT   M0093C	// RT_2D CODE TM OUT
AND NOT   M0093D	// RT_2D CODE NG
NOT
OR LOAD
MOVP      900 M0029
; L40
LOAD<>    0 M0092
MOVP      920 M0029
; L41
END

PROGRAM AUTO_LOAD (task: ¨ö¨¬A¥ì CA¡¤I¡¾¡¿¡¤¡Í)

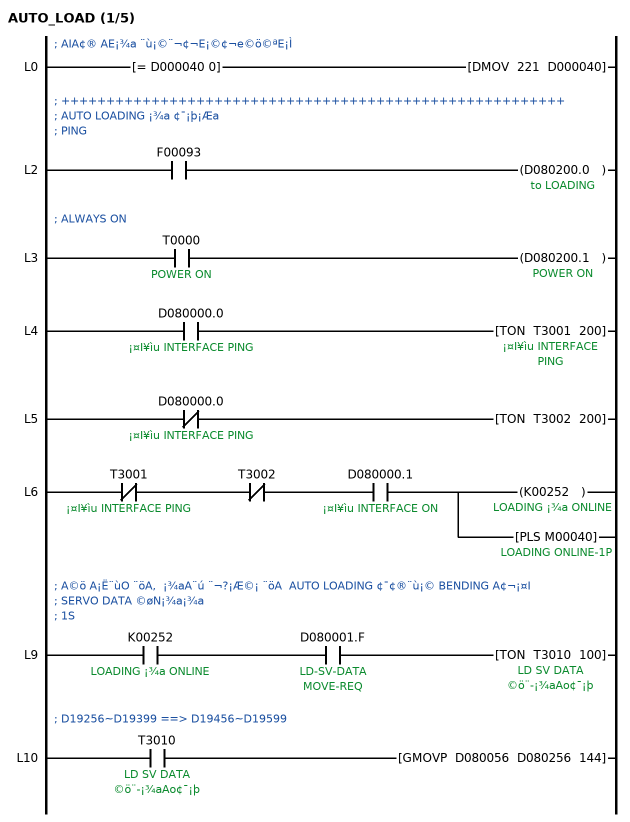
; L0
LOAD=     D000040 0
DMOV      221 D000040
// output comment: AIA¢® AE¡¾a ¨ù¡©¨¬¢¬E¡©¢¬e©ö©ªE¡Ì
// ++++++++++++++++++++++++++++++++++++++++++++++++++++++++
//    AUTO LOADING ¡¾a ¢¯¡þ¡Æa
; L2
LOAD      F00093
OUT       D080200.0	// to LOADING
// output comment: PING
; L3
LOAD      T0000	// POWER ON
OUT       D080200.1	// POWER ON
// output comment: ALWAYS ON
; L4
LOAD      D080000.0	// ¡¤I¥ìu INTERFACE PING
TON       T3001 200	// ¡¤I¥ìu INTERFACE PING
; L5
LOAD NOT  D080000.0	// ¡¤I¥ìu INTERFACE PING
TON       T3002 200
; L6
LOAD NOT  T3001	// ¡¤I¥ìu INTERFACE PING
AND NOT   T3002
AND       D080000.1	// ¡¤I¥ìu INTERFACE ON
OUT       K00252	// LOADING ¡¾a ONLINE
OUTP      M00040	// LOADING ONLINE-1P
// A©ö A¡Ë¨ùO ¨öA,  ¡¾aA¨ú ¨¬?¡Æ©¡ ¨öA  AUTO LOADING ¢¯¢®¨ù¡© BENDING A¢¬¡¤I  SERVO DATA ©øN¡¾a¡¾a
; L9
LOAD      K00252	// LOADING ¡¾a ONLINE
AND       D080001.F	// LD-SV-DATA MOVE-REQ
TON       T3010 100	// LD SV DATA ©ö¨­¡¾aAo¢¯¡þ
// output comment: 1S
; L10
LOAD      T3010	// LD SV DATA ©ö¨­¡¾aAo¢¯¡þ
GMOVP     D080056 D080256 144
// output comment: D19256~D19399 ==> D19456~D19599

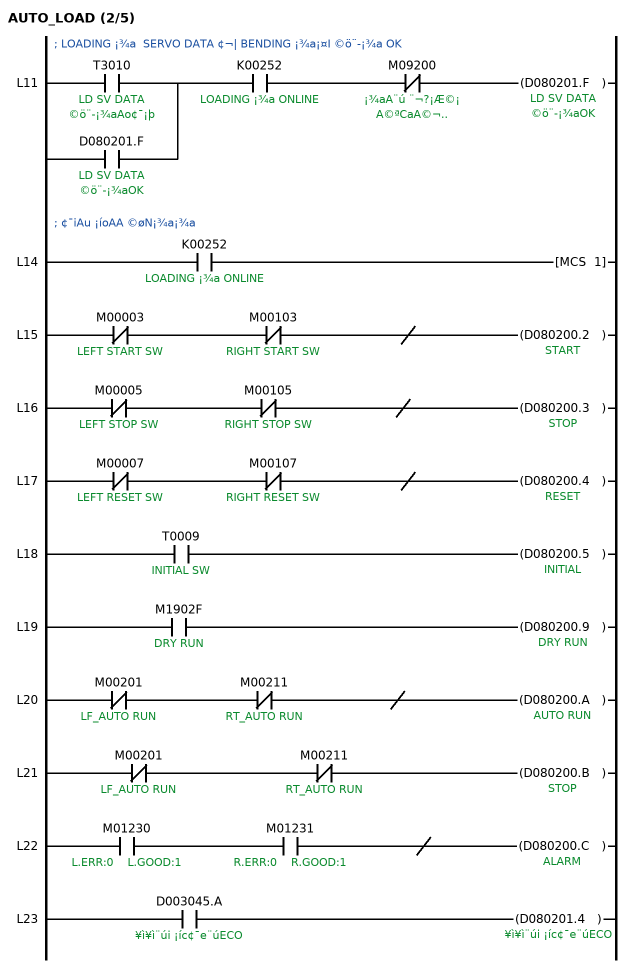
; L11
LOAD      T3010	// LD SV DATA ©ö¨­¡¾aAo¢¯¡þ
OR        D080201.F	// LD SV DATA ©ö¨­¡¾aOK
AND       K00252	// LOADING ¡¾a ONLINE
AND NOT   M09200	// ¡¾aA¨ú ¨¬?¡Æ©¡ A©ªCaA©¬..
OUT       D080201.F	// LD SV DATA ©ö¨­¡¾aOK
// output comment: LOADING ¡¾a  SERVO DATA ¢¬| BENDING ¡¾a¡¤I ©ö¨­¡¾a OK
// ¢¯iAu ¡íoAA ©øN¡¾a¡¾a
; L14
LOAD      K00252	// LOADING ¡¾a ONLINE
MCS       1
; L15
LOAD NOT  M00003	// LEFT START SW
AND NOT   M00103	// RIGHT START SW
NOT
OUT       D080200.2	// START
; L16
LOAD NOT  M00005	// LEFT STOP SW
AND NOT   M00105	// RIGHT STOP SW
NOT
OUT       D080200.3	// STOP
; L17
LOAD NOT  M00007	// LEFT RESET SW
AND NOT   M00107	// RIGHT RESET SW
NOT
OUT       D080200.4	// RESET
; L18
LOAD      T0009	// INITIAL SW
OUT       D080200.5	// INITIAL
; L19
LOAD      M1902F	// DRY RUN
OUT       D080200.9	// DRY RUN
; L20
LOAD NOT  M00201	// LF_AUTO RUN
AND NOT   M00211	// RT_AUTO RUN
NOT
OUT       D080200.A	// AUTO RUN
; L21
LOAD NOT  M00201	// LF_AUTO RUN
AND NOT   M00211	// RT_AUTO RUN
OUT       D080200.B	// STOP
; L22
LOAD      M01230	// L.ERR:0    L.GOOD:1
AND       M01231	// R.ERR:0    R.GOOD:1
NOT
OUT       D080200.C	// ALARM
; L23
LOAD      D003045.A	// ¥ì¥ì¨úi ¡íc¢¯e¨úECO
OUT       D080201.4	// ¥ì¥ì¨úi ¡íc¢¯e¨úECO

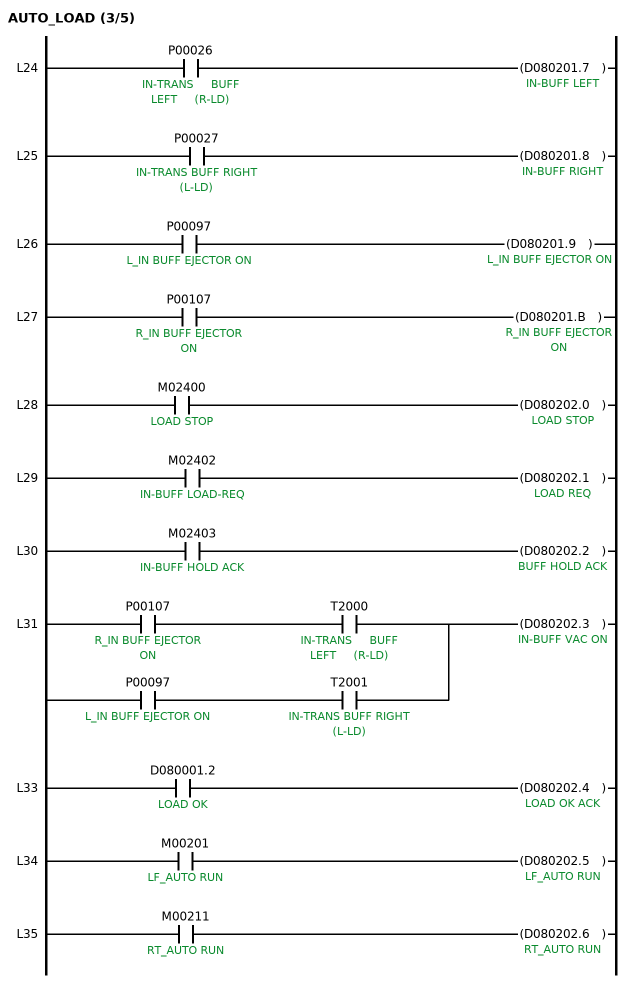
; L24
LOAD      P00026	// IN-TRANS     BUFF     LEFT     (R-LD)
OUT       D080201.7	// IN-BUFF LEFT
; L25
LOAD      P00027	// IN-TRANS BUFF RIGHT     (L-LD)
OUT       D080201.8	// IN-BUFF RIGHT
; L26
LOAD      P00097	// L_IN BUFF EJECTOR ON
OUT       D080201.9	// L_IN BUFF EJECTOR ON
; L27
LOAD      P00107	// R_IN BUFF EJECTOR ON
OUT       D080201.B	// R_IN BUFF EJECTOR ON
; L28
LOAD      M02400	// LOAD STOP
OUT       D080202.0	// LOAD STOP
; L29
LOAD      M02402	// IN-BUFF LOAD-REQ
OUT       D080202.1	// LOAD REQ
; L30
LOAD      M02403	// IN-BUFF HOLD ACK
OUT       D080202.2	// BUFF HOLD ACK
; L31
LOAD      P00107	// R_IN BUFF EJECTOR ON
AND       T2000	// IN-TRANS     BUFF     LEFT     (R-LD)
LOAD      P00097	// L_IN BUFF EJECTOR ON
AND       T2001	// IN-TRANS BUFF RIGHT     (L-LD)
OR LOAD
OUT       D080202.3	// IN-BUFF VAC ON
; L33
LOAD      D080001.2	// LOAD OK
OUT       D080202.4	// LOAD OK ACK
; L34
LOAD      M00201	// LF_AUTO RUN
OUT       D080202.5	// LF_AUTO RUN
; L35
LOAD      M00211	// RT_AUTO RUN
OUT       D080202.6	// RT_AUTO RUN

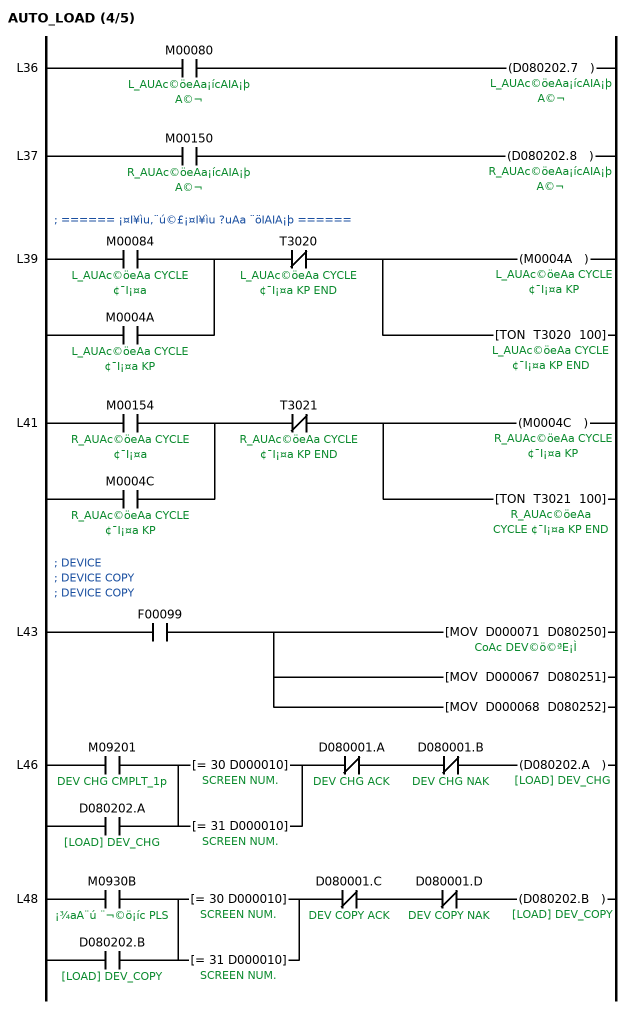
; L36
LOAD      M00080	// L_AUAc©öeAa¡ícAIA¡þA©¬
OUT       D080202.7	// L_AUAc©öeAa¡ícAIA¡þA©¬
; L37
LOAD      M00150	// R_AUAc©öeAa¡ícAIA¡þA©¬
OUT       D080202.8	// R_AUAc©öeAa¡ícAIA¡þA©¬
// ====== ¡¤I¥ìu,¨ú©£¡¤I¥ìu ?uAa ¨öIAIA¡þ ======
; L39
LOAD      M00084	// L_AUAc©öeAa CYCLE ¢¯I¡¤a
OR        M0004A	// L_AUAc©öeAa CYCLE ¢¯I¡¤a KP
AND NOT   T3020	// L_AUAc©öeAa CYCLE ¢¯I¡¤a KP END
OUT       M0004A	// L_AUAc©öeAa CYCLE ¢¯I¡¤a KP
TON       T3020 100	// L_AUAc©öeAa CYCLE ¢¯I¡¤a KP END
; L41
LOAD      M00154	// R_AUAc©öeAa CYCLE ¢¯I¡¤a
OR        M0004C	// R_AUAc©öeAa CYCLE ¢¯I¡¤a KP
AND NOT   T3021	// R_AUAc©öeAa CYCLE ¢¯I¡¤a KP END
OUT       M0004C	// R_AUAc©öeAa CYCLE ¢¯I¡¤a KP
TON       T3021 100	// R_AUAc©öeAa CYCLE ¢¯I¡¤a KP END
; L43
LOAD      F00099
MOV       D000071 D080250	// CoAc DEV©ö©ªE¡Ì
MOV       D000067 D080251
MOV       D000068 D080252
// output comment: DEVICE
// output comment: DEVICE COPY
// output comment: DEVICE COPY
; L46
LOAD      M09201	// DEV CHG CMPLT_1p
OR        D080202.A	// [LOAD] DEV_CHG
LOAD=     30 D000010	// SCREEN NUM.
OR=       31 D000010	// SCREEN NUM.
AND LOAD
AND NOT   D080001.A	// DEV CHG ACK
AND NOT   D080001.B	// DEV CHG NAK
OUT       D080202.A	// [LOAD] DEV_CHG
; L48
LOAD      M0930B	// ¡¾aA¨ú ¨¬©ö¡íc PLS
OR        D080202.B	// [LOAD] DEV_COPY
LOAD=     30 D000010	// SCREEN NUM.
OR=       31 D000010	// SCREEN NUM.
AND LOAD
AND NOT   D080001.C	// DEV COPY ACK
AND NOT   D080001.D	// DEV COPY NAK
OUT       D080202.B	// [LOAD] DEV_COPY

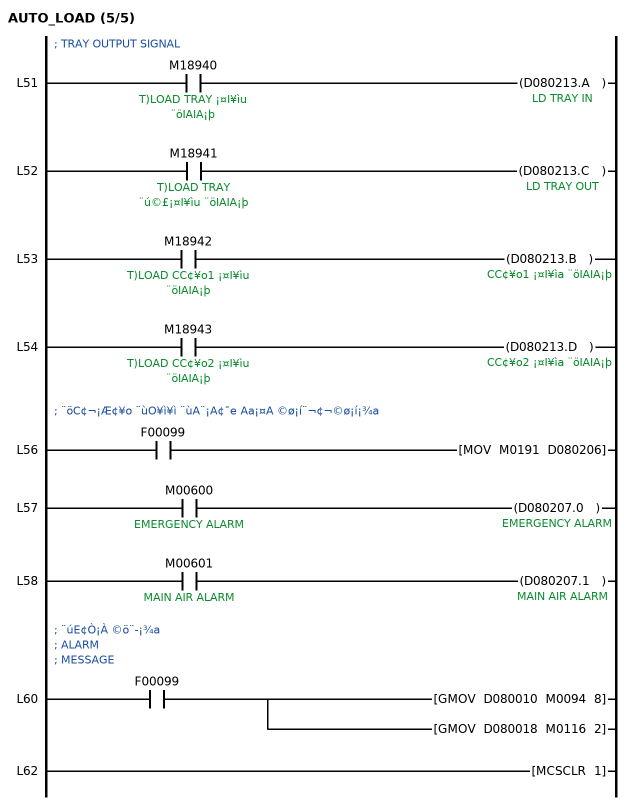
// TRAY OUTPUT SIGNAL
; L51
LOAD      M18940	// T)LOAD TRAY ¡¤I¥ìu ¨öIAIA¡þ
OUT       D080213.A	// LD TRAY IN
; L52
LOAD      M18941	// T)LOAD TRAY ¨ú©£¡¤I¥ìu ¨öIAIA¡þ
OUT       D080213.C	// LD TRAY OUT
; L53
LOAD      M18942	// T)LOAD CC¢¥o1 ¡¤I¥ìu ¨öIAIA¡þ
OUT       D080213.B	// CC¢¥o1 ¡¤I¥ìa ¨öIAIA¡þ
; L54
LOAD      M18943	// T)LOAD CC¢¥o2 ¡¤I¥ìu ¨öIAIA¡þ
OUT       D080213.D	// CC¢¥o2 ¡¤I¥ìa ¨öIAIA¡þ
// ¨öC¢¬¡Æ¢¥o ¨ùO¥ì¥ì ¨ùA¨¡A¢¯e Aa¡¤A ©ø¡í¨¬¢¬©ø¡í¡¾a
; L56
LOAD      F00099
MOV       M0191 D080206
; L57
LOAD      M00600	// EMERGENCY ALARM
OUT       D080207.0	// EMERGENCY ALARM
; L58
LOAD      M00601	// MAIN AIR ALARM
OUT       D080207.1	// MAIN AIR ALARM
// ¨úE¢Ò¡À ©ö¨­¡¾a
; L60
LOAD      F00099
GMOV      D080010 M0094 8
GMOV      D080018 M0116 2
// output comment: ALARM
// output comment: MESSAGE
; L62
MCSCLR    1

PROGRAM AUTO_UNLOAD (task: ¨ö¨¬A¥ì CA¡¤I¡¾¡¿¡¤¡Í)

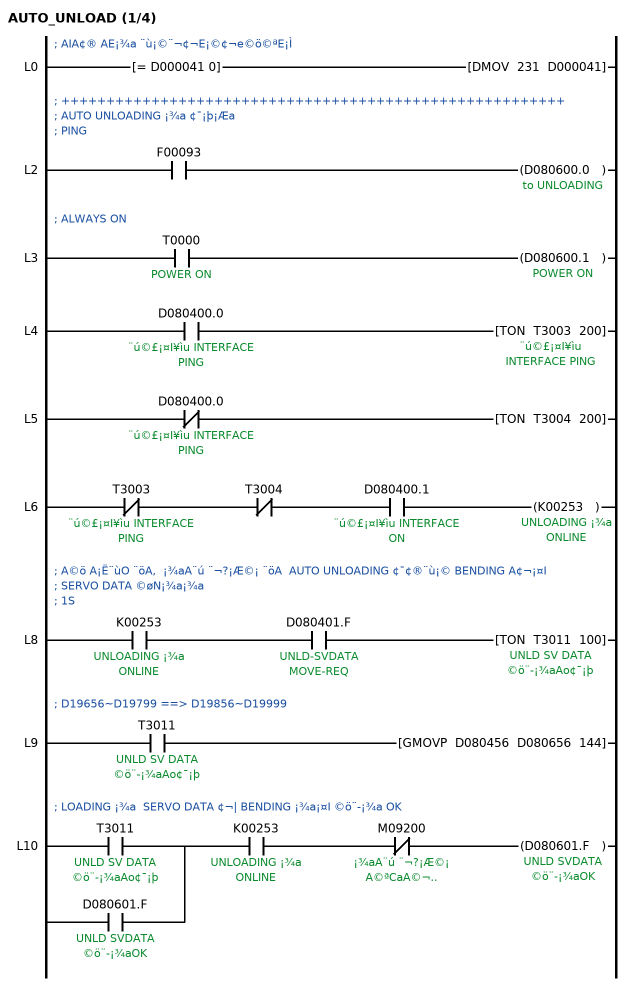
; L0
LOAD=     D000041 0
DMOV      231 D000041
// output comment: AIA¢® AE¡¾a ¨ù¡©¨¬¢¬E¡©¢¬e©ö©ªE¡Ì
// ++++++++++++++++++++++++++++++++++++++++++++++++++++++++
//    AUTO UNLOADING ¡¾a ¢¯¡þ¡Æa
; L2
LOAD      F00093
OUT       D080600.0	// to UNLOADING
// output comment: PING
; L3
LOAD      T0000	// POWER ON
OUT       D080600.1	// POWER ON
// output comment: ALWAYS ON
; L4
LOAD      D080400.0	// ¨ú©£¡¤I¥ìu INTERFACE PING
TON       T3003 200	// ¨ú©£¡¤I¥ìu INTERFACE PING
; L5
LOAD NOT  D080400.0	// ¨ú©£¡¤I¥ìu INTERFACE PING
TON       T3004 200
; L6
LOAD NOT  T3003	// ¨ú©£¡¤I¥ìu INTERFACE PING
AND NOT   T3004
AND       D080400.1	// ¨ú©£¡¤I¥ìu INTERFACE ON
OUT       K00253	// UNLOADING ¡¾a ONLINE
// A©ö A¡Ë¨ùO ¨öA,  ¡¾aA¨ú ¨¬?¡Æ©¡ ¨öA  AUTO UNLOADING ¢¯¢®¨ù¡© BENDING A¢¬¡¤I  SERVO DATA ©øN¡¾a¡¾a
; L8
LOAD      K00253	// UNLOADING ¡¾a ONLINE
AND       D080401.F	// UNLD-SVDATA MOVE-REQ
TON       T3011 100	// UNLD SV DATA ©ö¨­¡¾aAo¢¯¡þ
// output comment: 1S
; L9
LOAD      T3011	// UNLD SV DATA ©ö¨­¡¾aAo¢¯¡þ
GMOVP     D080456 D080656 144
// output comment: D19656~D19799 ==> D19856~D19999
; L10
LOAD      T3011	// UNLD SV DATA ©ö¨­¡¾aAo¢¯¡þ
OR        D080601.F	// UNLD SVDATA ©ö¨­¡¾aOK
AND       K00253	// UNLOADING ¡¾a ONLINE
AND NOT   M09200	// ¡¾aA¨ú ¨¬?¡Æ©¡ A©ªCaA©¬..
OUT       D080601.F	// UNLD SVDATA ©ö¨­¡¾aOK
// output comment: LOADING ¡¾a  SERVO DATA ¢¬| BENDING ¡¾a¡¤I ©ö¨­¡¾a OK

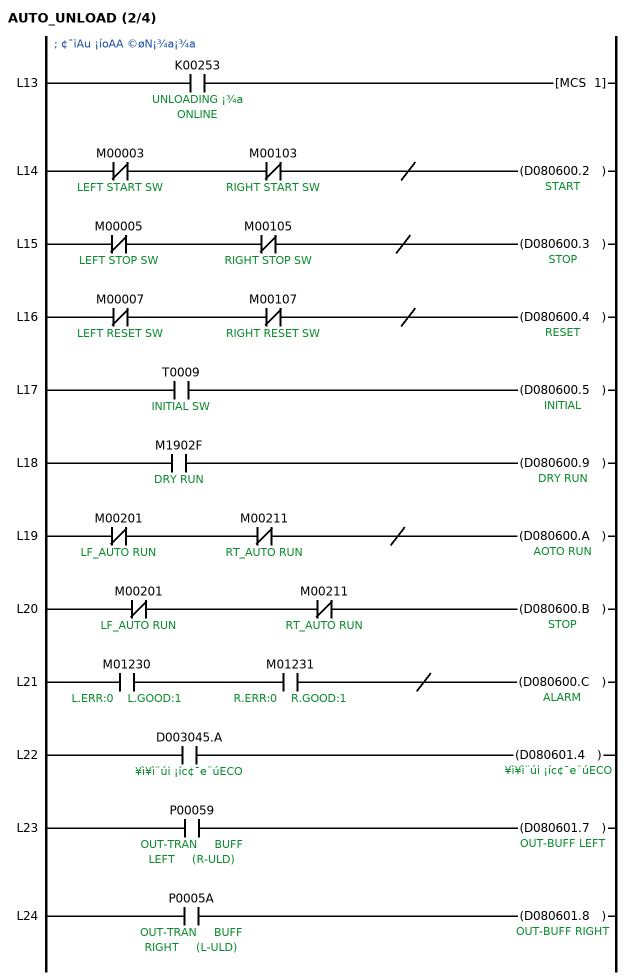
// ¢¯iAu ¡íoAA ©øN¡¾a¡¾a
; L13
LOAD      K00253	// UNLOADING ¡¾a ONLINE
MCS       1
; L14
LOAD NOT  M00003	// LEFT START SW
AND NOT   M00103	// RIGHT START SW
NOT
OUT       D080600.2	// START
; L15
LOAD NOT  M00005	// LEFT STOP SW
AND NOT   M00105	// RIGHT STOP SW
NOT
OUT       D080600.3	// STOP
; L16
LOAD NOT  M00007	// LEFT RESET SW
AND NOT   M00107	// RIGHT RESET SW
NOT
OUT       D080600.4	// RESET
; L17
LOAD      T0009	// INITIAL SW
OUT       D080600.5	// INITIAL
; L18
LOAD      M1902F	// DRY RUN
OUT       D080600.9	// DRY RUN
; L19
LOAD NOT  M00201	// LF_AUTO RUN
AND NOT   M00211	// RT_AUTO RUN
NOT
OUT       D080600.A	// AOTO RUN
; L20
LOAD NOT  M00201	// LF_AUTO RUN
AND NOT   M00211	// RT_AUTO RUN
OUT       D080600.B	// STOP
; L21
LOAD      M01230	// L.ERR:0    L.GOOD:1
AND       M01231	// R.ERR:0    R.GOOD:1
NOT
OUT       D080600.C	// ALARM
; L22
LOAD      D003045.A	// ¥ì¥ì¨úi ¡íc¢¯e¨úECO
OUT       D080601.4	// ¥ì¥ì¨úi ¡íc¢¯e¨úECO
; L23
LOAD      P00059	// OUT-TRAN     BUFF     LEFT     (R-ULD)
OUT       D080601.7	// OUT-BUFF LEFT
; L24
LOAD      P0005A	// OUT-TRAN     BUFF     RIGHT     (L-ULD)
OUT       D080601.8	// OUT-BUFF RIGHT

